	MoveL Offs(p0,26.0,100.0, 0), v10, z5, tool0;
	MoveL Offs(p0,27.0,102.0, 0), v10, z5, tool0;
	MoveL Offs(p0,27.0,104.0, 0), v10, z5, tool0;
	MoveL Offs(p0,27.0,107.0, 0), v10, z5, tool0;
	MoveL Offs(p0,27.0,109.0, 0), v10, z5, tool0;
	MoveL Offs(p0,27.0,110.0, 0), v10, z5, tool0;
	MoveL Offs(p0,26.0,112.0, 0), v10, z5, tool0;
	MoveL Offs(p0,26.0,113.0, 0), v10, z5, tool0;
	MoveL Offs(p0,29.0,114.0, 0), v10, z5, tool0;
	MoveJ Offs(p0,29.0,114.0, 20), v10, z1, tool0;
	MoveJ Offs(p0,123.0,112.0, 20), v10, z1, tool0;
	MoveJ Offs(p0,123.0,112.0, 0), v10, z1, tool0;
	MoveL Offs(p0,125.0,110.0, 0), v10, z5, tool0;
	MoveL Offs(p0,125.0,109.0, 0), v10, z5, tool0;
	MoveL Offs(p0,126.0,107.0, 0), v10, z5, tool0;
	MoveL Offs(p0,127.0,106.0, 0), v10, z5, tool0;
	MoveL Offs(p0,128.0,104.0, 0), v10, z5, tool0;
	MoveL Offs(p0,130.0,101.0, 0), v10, z5, tool0;
	MoveL Offs(p0,131.0,98.0, 0), v10, z5, tool0;
	MoveL Offs(p0,133.0,95.0, 0), v10, z5, tool0;
	MoveL Offs(p0,134.0,92.0, 0), v10, z5, tool0;
	MoveL Offs(p0,135.0,91.0, 0), v10, z5, tool0;
	MoveL Offs(p0,136.0,90.0, 0), v10, z5, tool0;
	MoveL Offs(p0,137.0,89.0, 0), v10, z5, tool0;
	MoveL Offs(p0,137.0,87.0, 0), v10, z5, tool0;
	MoveL Offs(p0,138.0,86.0, 0), v10, z5, tool0;
	MoveL Offs(p0,139.0,84.0, 0), v10, z5, tool0;
	MoveL Offs(p0,140.0,82.0, 0), v10, z5, tool0;
	MoveL Offs(p0,141.0,80.0, 0), v10, z5, tool0;
	MoveL Offs(p0,143.0,78.0, 0), v10, z5, tool0;
	MoveL Offs(p0,144.0,76.0, 0), v10, z5, tool0;
	MoveL Offs(p0,145.0,74.0, 0), v10, z5, tool0;
	MoveL Offs(p0,146.0,72.0, 0), v10, z5, tool0;
	MoveL Offs(p0,147.0,71.0, 0), v10, z5, tool0;
	MoveL Offs(p0,147.0,70.0, 0), v10, z5, tool0;
	MoveL Offs(p0,147.0,69.0, 0), v10, z5, tool0;
	MoveL Offs(p0,148.0,69.0, 0), v10, z5, tool0;
	MoveL Offs(p0,148.0,68.0, 0), v10, z5, tool0;
	MoveL Offs(p0,148.0,67.0, 0), v10, z5, tool0;
	MoveL Offs(p0,147.0,65.0, 0), v10, z5, tool0;
	MoveL Offs(p0,147.0,64.0, 0), v10, z5, tool0;
	MoveL Offs(p0,146.0,63.0, 0), v10, z5, tool0;
	MoveL Offs(p0,145.0,63.0, 0), v10, z5, tool0;
	MoveL Offs(p0,145.0,62.0, 0), v10, z5, tool0;
	MoveL Offs(p0,144.0,61.0, 0), v10, z5, tool0;
	MoveL Offs(p0,142.0,60.0, 0), v10, z5, tool0;
	MoveL Offs(p0,141.0,59.0, 0), v10, z5, tool0;
	MoveL Offs(p0,139.0,58.0, 0), v10, z5, tool0;
	MoveL Offs(p0,137.0,57.0, 0), v10, z5, tool0;
	MoveL Offs(p0,135.0,56.0, 0), v10, z5, tool0;
	MoveL Offs(p0,133.0,55.0, 0), v10, z5, tool0;
	MoveL Offs(p0,131.0,54.0, 0), v10, z5, tool0;
	MoveL Offs(p0,129.0,53.0, 0), v10, z5, tool0;
	MoveL Offs(p0,127.0,53.0, 0), v10, z5, tool0;
	MoveL Offs(p0,126.0,52.0, 0), v10, z5, tool0;
	MoveL Offs(p0,125.0,52.0, 0), v10, z5, tool0;
	MoveL Offs(p0,124.0,52.0, 0), v10, z5, tool0;
	MoveL Offs(p0,122.0,53.0, 0), v10, z5, tool0;
	MoveL Offs(p0,121.0,53.0, 0), v10, z5, tool0;
	MoveL Offs(p0,121.0,54.0, 0), v10, z5, tool0;
	MoveL Offs(p0,120.0,55.0, 0), v10, z5, tool0;
	MoveL Offs(p0,119.0,57.0, 0), v10, z5, tool0;
	MoveL Offs(p0,118.0,59.0, 0), v10, z5, tool0;
	MoveL Offs(p0,116.0,61.0, 0), v10, z5, tool0;
	MoveL Offs(p0,115.0,64.0, 0), v10, z5, tool0;
	MoveL Offs(p0,113.0,67.0, 0), v10, z5, tool0;
	MoveL Offs(p0,112.0,69.0, 0), v10, z5, tool0;
	MoveL Offs(p0,112.0,71.0, 0), v10, z5, tool0;
	MoveL Offs(p0,111.0,72.0, 0), v10, z5, tool0;
	MoveL Offs(p0,110.0,73.0, 0), v10, z5, tool0;
	MoveL Offs(p0,110.0,74.0, 0), v10, z5, tool0;
	MoveL Offs(p0,109.0,75.0, 0), v10, z5, tool0;
	MoveL Offs(p0,109.0,76.0, 0), v10, z5, tool0;
	MoveL Offs(p0,108.0,76.0, 0), v10, z5, tool0;
	MoveL Offs(p0,107.0,79.0, 0), v10, z5, tool0;
	MoveL Offs(p0,105.0,81.0, 0), v10, z5, tool0;
	MoveL Offs(p0,104.0,83.0, 0), v10, z5, tool0;
	MoveL Offs(p0,103.0,85.0, 0), v10, z5, tool0;
	MoveL Offs(p0,101.0,86.0, 0), v10, z5, tool0;
	MoveL Offs(p0,100.0,88.0, 0), v10, z5, tool0;
	MoveL Offs(p0,99.0,89.0, 0), v10, z5, tool0;
	MoveL Offs(p0,98.0,91.0, 0), v10, z5, tool0;
	MoveL Offs(p0,97.0,91.0, 0), v10, z5, tool0;
	MoveL Offs(p0,95.0,94.0, 0), v10, z5, tool0;
	MoveL Offs(p0,95.0,94.0, 0), v10, z5, tool0;
	MoveL Offs(p0,94.0,95.0, 0), v10, z5, tool0;
	MoveL Offs(p0,94.0,95.0, 0), v10, z5, tool0;
	MoveL Offs(p0,94.0,96.0, 0), v10, z5, tool0;
	MoveL Offs(p0,94.0,96.0, 0), v10, z5, tool0;
	MoveL Offs(p0,94.0,97.0, 0), v10, z5, tool0;
	MoveL Offs(p0,95.0,99.0, 0), v10, z5, tool0;
	MoveL Offs(p0,95.0,100.0, 0), v10, z5, tool0;
	MoveL Offs(p0,96.0,100.0, 0), v10, z5, tool0;
	MoveL Offs(p0,96.0,100.0, 0), v10, z5, tool0;
	MoveL Offs(p0,97.0,100.0, 0), v10, z5, tool0;
	MoveL Offs(p0,98.0,101.0, 0), v10, z5, tool0;
	MoveL Offs(p0,99.0,101.0, 0), v10, z5, tool0;
	MoveL Offs(p0,102.0,101.0, 0), v10, z5, tool0;
	MoveL Offs(p0,102.0,101.0, 0), v10, z5, tool0;
	MoveL Offs(p0,103.0,102.0, 0), v10, z5, tool0;
	MoveL Offs(p0,104.0,102.0, 0), v10, z5, tool0;
	MoveL Offs(p0,104.0,102.0, 0), v10, z5, tool0;
	MoveL Offs(p0,105.0,103.0, 0), v10, z5, tool0;
	MoveL Offs(p0,106.0,103.0, 0), v10, z5, tool0;
	MoveL Offs(p0,109.0,105.0, 0), v10, z5, tool0;
	MoveL Offs(p0,110.0,105.0, 0), v10, z5, tool0;
	MoveL Offs(p0,111.0,106.0, 0), v10, z5, tool0;
	MoveL Offs(p0,112.0,107.0, 0), v10, z5, tool0;
	MoveL Offs(p0,113.0,108.0, 0), v10, z5, tool0;
	MoveL Offs(p0,114.0,108.0, 0), v10, z5, tool0;
	MoveL Offs(p0,115.0,109.0, 0), v10, z5, tool0;
	MoveL Offs(p0,116.0,110.0, 0), v10, z5, tool0;
	MoveL Offs(p0,116.0,111.0, 0), v10, z5, tool0;
	MoveL Offs(p0,118.0,113.0, 0), v10, z5, tool0;
	MoveL Offs(p0,118.0,113.0, 0), v10, z5, tool0;
	MoveL Offs(p0,119.0,113.0, 0), v10, z5, tool0;
	MoveL Offs(p0,119.0,113.0, 0), v10, z5, tool0;
	MoveL Offs(p0,119.0,114.0, 0), v10, z5, tool0;
	MoveL Offs(p0,120.0,114.0, 0), v10, z5, tool0;
	MoveL Offs(p0,120.0,114.0, 0), v10, z5, tool0;
	MoveL Offs(p0,122.0,113.0, 0), v10, z5, tool0;
	MoveL Offs(p0,123.0,113.0, 0), v10, z5, tool0;
	MoveL Offs(p0,123.0,112.0, 0), v10, z5, tool0;
	MoveL Offs(p0,123.0,112.0, 0), v10, z5, tool0;
	MoveJ Offs(p0,123.0,112.0, 20), v10, z1, tool0;
	MoveJ Offs(p0,76.0,113.0, 20), v10, z1, tool0;
	MoveJ Offs(p0,76.0,113.0, 0), v10, z1, tool0;
	MoveL Offs(p0,75.0,109.0, 0), v10, z5, tool0;
	MoveL Offs(p0,74.0,109.0, 0), v10, z5, tool0;
	MoveL Offs(p0,74.0,108.0, 0), v10, z5, tool0;
	MoveL Offs(p0,73.0,107.0, 0), v10, z5, tool0;
	MoveL Offs(p0,72.0,107.0, 0), v10, z5, tool0;
	MoveL Offs(p0,71.0,106.0, 0), v10, z5, tool0;
	MoveL Offs(p0,69.0,104.0, 0), v10, z5, tool0;
	MoveL Offs(p0,69.0,104.0, 0), v10, z5, tool0;
	MoveL Offs(p0,68.0,104.0, 0), v10, z5, tool0;
	MoveL Offs(p0,68.0,104.0, 0), v10, z5, tool0;
	MoveL Offs(p0,67.0,104.0, 0), v10, z5, tool0;
	MoveL Offs(p0,67.0,104.0, 0), v10, z5, tool0;
	MoveL Offs(p0,67.0,105.0, 0), v10, z5, tool0;
	MoveL Offs(p0,66.0,105.0, 0), v10, z5, tool0;
	MoveL Offs(p0,65.0,106.0, 0), v10, z5, tool0;
	MoveL Offs(p0,69.0,109.0, 0), v10, z5, tool0;
	MoveL Offs(p0,71.0,111.0, 0), v10, z5, tool0;
	MoveL Offs(p0,72.0,112.0, 0), v10, z5, tool0;
	MoveL Offs(p0,72.0,112.0, 0), v10, z5, tool0;
	MoveL Offs(p0,72.0,112.0, 0), v10, z5, tool0;
	MoveL Offs(p0,73.0,113.0, 0), v10, z5, tool0;
	MoveL Offs(p0,73.0,113.0, 0), v10, z5, tool0;
	MoveL Offs(p0,73.0,113.0, 0), v10, z5, tool0;
	MoveL Offs(p0,76.0,113.0, 0), v10, z5, tool0;
	MoveJ Offs(p0,76.0,113.0, 20), v10, z1, tool0;
	MoveJ Offs(p0,116.0,113.0, 20), v10, z1, tool0;
	MoveJ Offs(p0,116.0,113.0, 0), v10, z1, tool0;
	MoveL Offs(p0,115.0,111.0, 0), v10, z5, tool0;
	MoveL Offs(p0,114.0,110.0, 0), v10, z5, tool0;
	MoveL Offs(p0,114.0,109.0, 0), v10, z5, tool0;
	MoveL Offs(p0,113.0,109.0, 0), v10, z5, tool0;
	MoveL Offs(p0,113.0,108.0, 0), v10, z5, tool0;
	MoveL Offs(p0,112.0,108.0, 0), v10, z5, tool0;
	MoveL Offs(p0,110.0,106.0, 0), v10, z5, tool0;
	MoveL Offs(p0,109.0,106.0, 0), v10, z5, tool0;
	MoveL Offs(p0,109.0,106.0, 0), v10, z5, tool0;
	MoveL Offs(p0,108.0,105.0, 0), v10, z5, tool0;
	MoveL Offs(p0,107.0,105.0, 0), v10, z5, tool0;
	MoveL Offs(p0,107.0,105.0, 0), v10, z5, tool0;
	MoveL Offs(p0,104.0,103.0, 0), v10, z5, tool0;
	MoveL Offs(p0,104.0,103.0, 0), v10, z5, tool0;
	MoveL Offs(p0,103.0,103.0, 0), v10, z5, tool0;
	MoveL Offs(p0,102.0,103.0, 0), v10, z5, tool0;
	MoveL Offs(p0,102.0,102.0, 0), v10, z5, tool0;
	MoveL Offs(p0,101.0,102.0, 0), v10, z5, tool0;
	MoveL Offs(p0,101.0,102.0, 0), v10, z5, tool0;
	MoveL Offs(p0,100.0,102.0, 0), v10, z5, tool0;
	MoveL Offs(p0,98.0,102.0, 0), v10, z5, tool0;
	MoveL Offs(p0,98.0,102.0, 0), v10, z5, tool0;
	MoveL Offs(p0,97.0,102.0, 0), v10, z5, tool0;
	MoveL Offs(p0,97.0,102.0, 0), v10, z5, tool0;
	MoveL Offs(p0,97.0,102.0, 0), v10, z5, tool0;
	MoveL Offs(p0,97.0,102.0, 0), v10, z5, tool0;
	MoveL Offs(p0,96.0,101.0, 0), v10, z5, tool0;
	MoveL Offs(p0,96.0,103.0, 0), v10, z5, tool0;
	MoveL Offs(p0,97.0,105.0, 0), v10, z5, tool0;
	MoveL Offs(p0,97.0,106.0, 0), v10, z5, tool0;
	MoveL Offs(p0,97.0,106.0, 0), v10, z5, tool0;
	MoveL Offs(p0,97.0,106.0, 0), v10, z5, tool0;
	MoveL Offs(p0,97.0,106.0, 0), v10, z5, tool0;
	MoveL Offs(p0,98.0,107.0, 0), v10, z5, tool0;
	MoveL Offs(p0,100.0,107.0, 0), v10, z5, tool0;
	MoveL Offs(p0,100.0,107.0, 0), v10, z5, tool0;
	MoveL Offs(p0,101.0,107.0, 0), v10, z5, tool0;
	MoveL Offs(p0,101.0,107.0, 0), v10, z5, tool0;
	MoveL Offs(p0,103.0,107.0, 0), v10, z5, tool0;
	MoveL Offs(p0,104.0,107.0, 0), v10, z5, tool0;
	MoveL Offs(p0,105.0,107.0, 0), v10, z5, tool0;
	MoveL Offs(p0,105.0,107.0, 0), v10, z5, tool0;
	MoveL Offs(p0,106.0,108.0, 0), v10, z5, tool0;
	MoveL Offs(p0,106.0,108.0, 0), v10, z5, tool0;
	MoveL Offs(p0,107.0,109.0, 0), v10, z5, tool0;
	MoveL Offs(p0,107.0,110.0, 0), v10, z5, tool0;
	MoveL Offs(p0,108.0,111.0, 0), v10, z5, tool0;
	MoveL Offs(p0,109.0,113.0, 0), v10, z5, tool0;
	MoveL Offs(p0,112.0,113.0, 0), v10, z5, tool0;
	MoveL Offs(p0,114.0,113.0, 0), v10, z5, tool0;
	MoveL Offs(p0,115.0,113.0, 0), v10, z5, tool0;
	MoveL Offs(p0,115.0,113.0, 0), v10, z5, tool0;
	MoveL Offs(p0,115.0,113.0, 0), v10, z5, tool0;
	MoveL Offs(p0,116.0,113.0, 0), v10, z5, tool0;
	MoveL Offs(p0,116.0,113.0, 0), v10, z5, tool0;
	MoveL Offs(p0,116.0,113.0, 0), v10, z5, tool0;
	MoveL Offs(p0,116.0,113.0, 0), v10, z5, tool0;
	MoveJ Offs(p0,116.0,113.0, 20), v10, z1, tool0;
	MoveJ Offs(p0,82.0,111.0, 20), v10, z1, tool0;
	MoveJ Offs(p0,82.0,111.0, 0), v10, z1, tool0;
	MoveL Offs(p0,84.0,110.0, 0), v10, z5, tool0;
	MoveL Offs(p0,84.0,109.0, 0), v10, z5, tool0;
	MoveL Offs(p0,85.0,109.0, 0), v10, z5, tool0;
	MoveL Offs(p0,86.0,106.0, 0), v10, z5, tool0;
	MoveL Offs(p0,87.0,105.0, 0), v10, z5, tool0;
	MoveL Offs(p0,88.0,104.0, 0), v10, z5, tool0;
	MoveL Offs(p0,89.0,103.0, 0), v10, z5, tool0;
	MoveL Offs(p0,90.0,103.0, 0), v10, z5, tool0;
	MoveL Offs(p0,91.0,102.0, 0), v10, z5, tool0;
	MoveL Offs(p0,92.0,102.0, 0), v10, z5, tool0;
	MoveL Offs(p0,93.0,102.0, 0), v10, z5, tool0;
	MoveL Offs(p0,94.0,102.0, 0), v10, z5, tool0;
	MoveL Offs(p0,94.0,100.0, 0), v10, z5, tool0;
	MoveL Offs(p0,94.0,100.0, 0), v10, z5, tool0;
	MoveL Offs(p0,93.0,98.0, 0), v10, z5, tool0;
	MoveL Offs(p0,93.0,97.0, 0), v10, z5, tool0;
	MoveL Offs(p0,93.0,96.0, 0), v10, z5, tool0;
	MoveL Offs(p0,93.0,96.0, 0), v10, z5, tool0;
	MoveL Offs(p0,93.0,95.0, 0), v10, z5, tool0;
	MoveL Offs(p0,93.0,95.0, 0), v10, z5, tool0;
	MoveL Offs(p0,93.0,94.0, 0), v10, z5, tool0;
	MoveL Offs(p0,95.0,92.0, 0), v10, z5, tool0;
	MoveL Offs(p0,95.0,91.0, 0), v10, z5, tool0;
	MoveL Offs(p0,96.0,91.0, 0), v10, z5, tool0;
	MoveL Offs(p0,96.0,90.0, 0), v10, z5, tool0;
	MoveL Offs(p0,97.0,90.0, 0), v10, z5, tool0;
	MoveL Offs(p0,99.0,88.0, 0), v10, z5, tool0;
	MoveL Offs(p0,99.0,87.0, 0), v10, z5, tool0;
	MoveL Offs(p0,100.0,86.0, 0), v10, z5, tool0;
	MoveL Offs(p0,101.0,86.0, 0), v10, z5, tool0;
	MoveL Offs(p0,101.0,85.0, 0), v10, z5, tool0;
	MoveL Offs(p0,102.0,84.0, 0), v10, z5, tool0;
	MoveL Offs(p0,102.0,84.0, 0), v10, z5, tool0;
	MoveL Offs(p0,102.0,83.0, 0), v10, z5, tool0;
	MoveL Offs(p0,95.0,86.0, 0), v10, z5, tool0;
	MoveL Offs(p0,95.0,86.0, 0), v10, z5, tool0;
	MoveL Offs(p0,94.0,86.0, 0), v10, z5, tool0;
	MoveL Offs(p0,93.0,86.0, 0), v10, z5, tool0;
	MoveL Offs(p0,93.0,86.0, 0), v10, z5, tool0;
	MoveL Offs(p0,92.0,86.0, 0), v10, z5, tool0;
	MoveL Offs(p0,92.0,85.0, 0), v10, z5, tool0;
	MoveL Offs(p0,89.0,85.0, 0), v10, z5, tool0;
	MoveL Offs(p0,88.0,84.0, 0), v10, z5, tool0;
	MoveL Offs(p0,87.0,84.0, 0), v10, z5, tool0;
	MoveL Offs(p0,87.0,84.0, 0), v10, z5, tool0;
	MoveL Offs(p0,86.0,84.0, 0), v10, z5, tool0;
	MoveL Offs(p0,86.0,84.0, 0), v10, z5, tool0;
	MoveL Offs(p0,85.0,85.0, 0), v10, z5, tool0;
	MoveL Offs(p0,85.0,85.0, 0), v10, z5, tool0;
	MoveL Offs(p0,84.0,86.0, 0), v10, z5, tool0;
	MoveL Offs(p0,84.0,87.0, 0), v10, z5, tool0;
	MoveL Offs(p0,85.0,88.0, 0), v10, z5, tool0;
	MoveL Offs(p0,86.0,90.0, 0), v10, z5, tool0;
	MoveL Offs(p0,86.0,91.0, 0), v10, z5, tool0;
	MoveL Offs(p0,86.0,91.0, 0), v10, z5, tool0;
	MoveL Offs(p0,86.0,92.0, 0), v10, z5, tool0;
	MoveL Offs(p0,86.0,92.0, 0), v10, z5, tool0;
	MoveL Offs(p0,85.0,93.0, 0), v10, z5, tool0;
	MoveL Offs(p0,84.0,95.0, 0), v10, z5, tool0;
	MoveL Offs(p0,83.0,96.0, 0), v10, z5, tool0;
	MoveL Offs(p0,82.0,96.0, 0), v10, z5, tool0;
	MoveL Offs(p0,81.0,97.0, 0), v10, z5, tool0;
	MoveL Offs(p0,79.0,97.0, 0), v10, z5, tool0;
	MoveL Offs(p0,78.0,97.0, 0), v10, z5, tool0;
	MoveL Offs(p0,76.0,97.0, 0), v10, z5, tool0;
	MoveL Offs(p0,74.0,97.0, 0), v10, z5, tool0;
	MoveL Offs(p0,72.0,97.0, 0), v10, z5, tool0;
	MoveL Offs(p0,68.0,96.0, 0), v10, z5, tool0;
	MoveL Offs(p0,67.0,97.0, 0), v10, z5, tool0;
	MoveL Offs(p0,66.0,99.0, 0), v10, z5, tool0;
	MoveL Offs(p0,66.0,100.0, 0), v10, z5, tool0;
	MoveL Offs(p0,66.0,100.0, 0), v10, z5, tool0;
	MoveL Offs(p0,67.0,101.0, 0), v10, z5, tool0;
	MoveL Offs(p0,67.0,101.0, 0), v10, z5, tool0;
	MoveL Offs(p0,68.0,102.0, 0), v10, z5, tool0;
	MoveL Offs(p0,70.0,103.0, 0), v10, z5, tool0;
	MoveL Offs(p0,71.0,104.0, 0), v10, z5, tool0;
	MoveL Offs(p0,73.0,105.0, 0), v10, z5, tool0;
	MoveL Offs(p0,74.0,106.0, 0), v10, z5, tool0;
	MoveL Offs(p0,75.0,108.0, 0), v10, z5, tool0;
	MoveL Offs(p0,76.0,109.0, 0), v10, z5, tool0;
	MoveL Offs(p0,77.0,110.0, 0), v10, z5, tool0;
	MoveL Offs(p0,77.0,110.0, 0), v10, z5, tool0;
	MoveL Offs(p0,78.0,111.0, 0), v10, z5, tool0;
	MoveL Offs(p0,82.0,111.0, 0), v10, z5, tool0;
	MoveL Offs(p0,82.0,111.0, 0), v10, z5, tool0;
	MoveL Offs(p0,82.0,111.0, 0), v10, z5, tool0;
	MoveJ Offs(p0,82.0,111.0, 20), v10, z1, tool0;
	MoveJ Offs(p0,62.0,110.0, 20), v10, z1, tool0;
	MoveJ Offs(p0,62.0,110.0, 0), v10, z1, tool0;
	MoveL Offs(p0,63.0,108.0, 0), v10, z5, tool0;
	MoveL Offs(p0,64.0,107.0, 0), v10, z5, tool0;
	MoveL Offs(p0,64.0,107.0, 0), v10, z5, tool0;
	MoveL Offs(p0,64.0,107.0, 0), v10, z5, tool0;
	MoveL Offs(p0,64.0,106.0, 0), v10, z5, tool0;
	MoveL Offs(p0,66.0,104.0, 0), v10, z5, tool0;
	MoveL Offs(p0,66.0,104.0, 0), v10, z5, tool0;
	MoveL Offs(p0,66.0,103.0, 0), v10, z5, tool0;
	MoveL Offs(p0,66.0,103.0, 0), v10, z5, tool0;
	MoveL Offs(p0,66.0,103.0, 0), v10, z5, tool0;
	MoveL Offs(p0,66.0,103.0, 0), v10, z5, tool0;
	MoveL Offs(p0,64.0,99.0, 0), v10, z5, tool0;
	MoveL Offs(p0,65.0,99.0, 0), v10, z5, tool0;
	MoveL Offs(p0,65.0,98.0, 0), v10, z5, tool0;
	MoveL Offs(p0,65.0,98.0, 0), v10, z5, tool0;
	MoveL Offs(p0,65.0,97.0, 0), v10, z5, tool0;
	MoveL Offs(p0,66.0,95.0, 0), v10, z5, tool0;
	MoveL Offs(p0,66.0,95.0, 0), v10, z5, tool0;
	MoveL Offs(p0,65.0,94.0, 0), v10, z5, tool0;
	MoveL Offs(p0,65.0,94.0, 0), v10, z5, tool0;
	MoveL Offs(p0,65.0,94.0, 0), v10, z5, tool0;
	MoveL Offs(p0,64.0,94.0, 0), v10, z5, tool0;
	MoveL Offs(p0,62.0,94.0, 0), v10, z5, tool0;
	MoveL Offs(p0,62.0,94.0, 0), v10, z5, tool0;
	MoveL Offs(p0,62.0,94.0, 0), v10, z5, tool0;
	MoveL Offs(p0,60.0,97.0, 0), v10, z5, tool0;
	MoveL Offs(p0,60.0,98.0, 0), v10, z5, tool0;
	MoveL Offs(p0,60.0,99.0, 0), v10, z5, tool0;
	MoveL Offs(p0,60.0,100.0, 0), v10, z5, tool0;
	MoveL Offs(p0,60.0,101.0, 0), v10, z5, tool0;
	MoveL Offs(p0,60.0,102.0, 0), v10, z5, tool0;
	MoveL Offs(p0,60.0,103.0, 0), v10, z5, tool0;
	MoveL Offs(p0,60.0,105.0, 0), v10, z5, tool0;
	MoveL Offs(p0,60.0,106.0, 0), v10, z5, tool0;
	MoveL Offs(p0,60.0,108.0, 0), v10, z5, tool0;
	MoveL Offs(p0,60.0,109.0, 0), v10, z5, tool0;
	MoveL Offs(p0,60.0,109.0, 0), v10, z5, tool0;
	MoveL Offs(p0,61.0,110.0, 0), v10, z5, tool0;
	MoveL Offs(p0,61.0,111.0, 0), v10, z5, tool0;
	MoveL Offs(p0,61.0,111.0, 0), v10, z5, tool0;
	MoveL Offs(p0,61.0,111.0, 0), v10, z5, tool0;
	MoveL Offs(p0,62.0,110.0, 0), v10, z5, tool0;
	MoveJ Offs(p0,62.0,110.0, 20), v10, z1, tool0;
	MoveJ Offs(p0,92.0,108.0, 20), v10, z1, tool0;
	MoveJ Offs(p0,92.0,108.0, 0), v10, z1, tool0;
	MoveL Offs(p0,93.0,106.0, 0), v10, z5, tool0;
	MoveL Offs(p0,93.0,106.0, 0), v10, z5, tool0;
	MoveL Offs(p0,93.0,106.0, 0), v10, z5, tool0;
	MoveL Offs(p0,91.0,103.0, 0), v10, z5, tool0;
	MoveL Offs(p0,89.0,105.0, 0), v10, z5, tool0;
	MoveL Offs(p0,88.0,106.0, 0), v10, z5, tool0;
	MoveL Offs(p0,88.0,106.0, 0), v10, z5, tool0;
	MoveL Offs(p0,87.0,107.0, 0), v10, z5, tool0;
	MoveL Offs(p0,87.0,107.0, 0), v10, z5, tool0;
	MoveL Offs(p0,86.0,108.0, 0), v10, z5, tool0;
	MoveL Offs(p0,85.0,110.0, 0), v10, z5, tool0;
	MoveL Offs(p0,86.0,110.0, 0), v10, z5, tool0;
	MoveL Offs(p0,86.0,110.0, 0), v10, z5, tool0;
	MoveL Offs(p0,87.0,110.0, 0), v10, z5, tool0;
	MoveL Offs(p0,87.0,110.0, 0), v10, z5, tool0;
	MoveL Offs(p0,91.0,110.0, 0), v10, z5, tool0;
	MoveL Offs(p0,91.0,109.0, 0), v10, z5, tool0;
	MoveL Offs(p0,91.0,109.0, 0), v10, z5, tool0;
	MoveL Offs(p0,91.0,109.0, 0), v10, z5, tool0;
	MoveL Offs(p0,91.0,109.0, 0), v10, z5, tool0;
	MoveL Offs(p0,91.0,109.0, 0), v10, z5, tool0;
	MoveL Offs(p0,92.0,108.0, 0), v10, z5, tool0;
	MoveL Offs(p0,92.0,108.0, 0), v10, z5, tool0;
	MoveJ Offs(p0,92.0,108.0, 20), v10, z1, tool0;
	MoveJ Offs(p0,146.0,98.0, 20), v10, z1, tool0;
	MoveJ Offs(p0,146.0,98.0, 0), v10, z1, tool0;
	MoveL Offs(p0,148.0,96.0, 0), v10, z5, tool0;
	MoveL Offs(p0,149.0,95.0, 0), v10, z5, tool0;
	MoveL Offs(p0,150.0,94.0, 0), v10, z5, tool0;
	MoveL Offs(p0,150.0,94.0, 0), v10, z5, tool0;
	MoveL Offs(p0,151.0,93.0, 0), v10, z5, tool0;
	MoveL Offs(p0,151.0,92.0, 0), v10, z5, tool0;
	MoveL Offs(p0,152.0,90.0, 0), v10, z5, tool0;
	MoveL Offs(p0,152.0,89.0, 0), v10, z5, tool0;
	MoveL Offs(p0,153.0,86.0, 0), v10, z5, tool0;
	MoveL Offs(p0,154.0,83.0, 0), v10, z5, tool0;
	MoveL Offs(p0,155.0,81.0, 0), v10, z5, tool0;
	MoveL Offs(p0,156.0,79.0, 0), v10, z5, tool0;
	MoveL Offs(p0,157.0,77.0, 0), v10, z5, tool0;
	MoveL Offs(p0,158.0,75.0, 0), v10, z5, tool0;
	MoveL Offs(p0,159.0,74.0, 0), v10, z5, tool0;
	MoveL Offs(p0,161.0,73.0, 0), v10, z5, tool0;
	MoveL Offs(p0,162.0,71.0, 0), v10, z5, tool0;
	MoveL Offs(p0,163.0,70.0, 0), v10, z5, tool0;
	MoveL Offs(p0,166.0,69.0, 0), v10, z5, tool0;
	MoveL Offs(p0,167.0,69.0, 0), v10, z5, tool0;
	MoveL Offs(p0,168.0,68.0, 0), v10, z5, tool0;
	MoveL Offs(p0,170.0,68.0, 0), v10, z5, tool0;
	MoveL Offs(p0,171.0,68.0, 0), v10, z5, tool0;
	MoveL Offs(p0,173.0,68.0, 0), v10, z5, tool0;
	MoveL Offs(p0,174.0,68.0, 0), v10, z5, tool0;
	MoveL Offs(p0,176.0,68.0, 0), v10, z5, tool0;
	MoveL Offs(p0,177.0,68.0, 0), v10, z5, tool0;
	MoveL Offs(p0,180.0,69.0, 0), v10, z5, tool0;
	MoveL Offs(p0,182.0,70.0, 0), v10, z5, tool0;
	MoveL Offs(p0,183.0,71.0, 0), v10, z5, tool0;
	MoveL Offs(p0,184.0,73.0, 0), v10, z5, tool0;
	MoveL Offs(p0,184.0,74.0, 0), v10, z5, tool0;
	MoveL Offs(p0,185.0,75.0, 0), v10, z5, tool0;
	MoveL Offs(p0,185.0,77.0, 0), v10, z5, tool0;
	MoveL Offs(p0,185.0,79.0, 0), v10, z5, tool0;
	MoveL Offs(p0,184.0,80.0, 0), v10, z5, tool0;
	MoveL Offs(p0,182.0,84.0, 0), v10, z5, tool0;
	MoveL Offs(p0,181.0,86.0, 0), v10, z5, tool0;
	MoveL Offs(p0,180.0,87.0, 0), v10, z5, tool0;
	MoveL Offs(p0,178.0,88.0, 0), v10, z5, tool0;
	MoveL Offs(p0,176.0,89.0, 0), v10, z5, tool0;
	MoveL Offs(p0,174.0,90.0, 0), v10, z5, tool0;
	MoveL Offs(p0,172.0,91.0, 0), v10, z5, tool0;
	MoveL Offs(p0,170.0,91.0, 0), v10, z5, tool0;
	MoveL Offs(p0,167.0,91.0, 0), v10, z5, tool0;
	MoveL Offs(p0,165.0,91.0, 0), v10, z5, tool0;
	MoveL Offs(p0,165.0,91.0, 0), v10, z5, tool0;
	MoveL Offs(p0,165.0,91.0, 0), v10, z5, tool0;
	MoveL Offs(p0,164.0,91.0, 0), v10, z5, tool0;
	MoveL Offs(p0,164.0,91.0, 0), v10, z5, tool0;
	MoveL Offs(p0,164.0,91.0, 0), v10, z5, tool0;
	MoveL Offs(p0,167.0,92.0, 0), v10, z5, tool0;
	MoveL Offs(p0,167.0,92.0, 0), v10, z5, tool0;
	MoveL Offs(p0,168.0,92.0, 0), v10, z5, tool0;
	MoveL Offs(p0,168.0,92.0, 0), v10, z5, tool0;
	MoveL Offs(p0,169.0,92.0, 0), v10, z5, tool0;
	MoveL Offs(p0,171.0,92.0, 0), v10, z5, tool0;
	MoveL Offs(p0,172.0,92.0, 0), v10, z5, tool0;
	MoveL Offs(p0,173.0,92.0, 0), v10, z5, tool0;
	MoveL Offs(p0,173.0,92.0, 0), v10, z5, tool0;
	MoveL Offs(p0,174.0,91.0, 0), v10, z5, tool0;
	MoveL Offs(p0,174.0,91.0, 0), v10, z5, tool0;
	MoveL Offs(p0,175.0,91.0, 0), v10, z5, tool0;
	MoveL Offs(p0,176.0,91.0, 0), v10, z5, tool0;
	MoveL Offs(p0,177.0,90.0, 0), v10, z5, tool0;
	MoveL Offs(p0,179.0,89.0, 0), v10, z5, tool0;
	MoveL Offs(p0,180.0,88.0, 0), v10, z5, tool0;
	MoveL Offs(p0,181.0,87.0, 0), v10, z5, tool0;
	MoveL Offs(p0,182.0,87.0, 0), v10, z5, tool0;
	MoveL Offs(p0,183.0,86.0, 0), v10, z5, tool0;
	MoveL Offs(p0,184.0,85.0, 0), v10, z5, tool0;
	MoveL Offs(p0,184.0,84.0, 0), v10, z5, tool0;
	MoveL Offs(p0,185.0,83.0, 0), v10, z5, tool0;
	MoveL Offs(p0,186.0,82.0, 0), v10, z5, tool0;
	MoveL Offs(p0,187.0,79.0, 0), v10, z5, tool0;
	MoveL Offs(p0,187.0,79.0, 0), v10, z5, tool0;
	MoveL Offs(p0,187.0,78.0, 0), v10, z5, tool0;
	MoveL Offs(p0,187.0,77.0, 0), v10, z5, tool0;
	MoveL Offs(p0,187.0,76.0, 0), v10, z5, tool0;
	MoveL Offs(p0,187.0,75.0, 0), v10, z5, tool0;
	MoveL Offs(p0,187.0,74.0, 0), v10, z5, tool0;
	MoveL Offs(p0,187.0,74.0, 0), v10, z5, tool0;
	MoveL Offs(p0,186.0,71.0, 0), v10, z5, tool0;
	MoveL Offs(p0,185.0,70.0, 0), v10, z5, tool0;
	MoveL Offs(p0,184.0,70.0, 0), v10, z5, tool0;
	MoveL Offs(p0,184.0,69.0, 0), v10, z5, tool0;
	MoveL Offs(p0,183.0,68.0, 0), v10, z5, tool0;
	MoveL Offs(p0,182.0,68.0, 0), v10, z5, tool0;
	MoveL Offs(p0,181.0,67.0, 0), v10, z5, tool0;
	MoveL Offs(p0,181.0,67.0, 0), v10, z5, tool0;
	MoveL Offs(p0,178.0,66.0, 0), v10, z5, tool0;
	MoveL Offs(p0,178.0,66.0, 0), v10, z5, tool0;
	MoveL Offs(p0,177.0,65.0, 0), v10, z5, tool0;
	MoveL Offs(p0,177.0,65.0, 0), v10, z5, tool0;
	MoveL Offs(p0,176.0,65.0, 0), v10, z5, tool0;
	MoveL Offs(p0,175.0,65.0, 0), v10, z5, tool0;
	MoveL Offs(p0,174.0,65.0, 0), v10, z5, tool0;
	MoveL Offs(p0,172.0,65.0, 0), v10, z5, tool0;
	MoveL Offs(p0,171.0,65.0, 0), v10, z5, tool0;
	MoveL Offs(p0,171.0,65.0, 0), v10, z5, tool0;
	MoveL Offs(p0,170.0,65.0, 0), v10, z5, tool0;
	MoveL Offs(p0,170.0,65.0, 0), v10, z5, tool0;
	MoveL Offs(p0,169.0,66.0, 0), v10, z5, tool0;
	MoveL Offs(p0,168.0,66.0, 0), v10, z5, tool0;
	MoveL Offs(p0,168.0,66.0, 0), v10, z5, tool0;
	MoveL Offs(p0,165.0,67.0, 0), v10, z5, tool0;
	MoveL Offs(p0,163.0,68.0, 0), v10, z5, tool0;
	MoveL Offs(p0,161.0,69.0, 0), v10, z5, tool0;
	MoveL Offs(p0,159.0,71.0, 0), v10, z5, tool0;
	MoveL Offs(p0,158.0,73.0, 0), v10, z5, tool0;
	MoveL Offs(p0,156.0,75.0, 0), v10, z5, tool0;
	MoveL Offs(p0,154.0,77.0, 0), v10, z5, tool0;
	MoveL Offs(p0,153.0,80.0, 0), v10, z5, tool0;
	MoveL Offs(p0,152.0,83.0, 0), v10, z5, tool0;
	MoveL Offs(p0,151.0,86.0, 0), v10, z5, tool0;
	MoveL Offs(p0,150.0,88.0, 0), v10, z5, tool0;
	MoveL Offs(p0,150.0,89.0, 0), v10, z5, tool0;
	MoveL Offs(p0,149.0,90.0, 0), v10, z5, tool0;
	MoveL Offs(p0,149.0,90.0, 0), v10, z5, tool0;
	MoveL Offs(p0,149.0,91.0, 0), v10, z5, tool0;
	MoveL Offs(p0,149.0,91.0, 0), v10, z5, tool0;
	MoveL Offs(p0,149.0,92.0, 0), v10, z5, tool0;
	MoveL Offs(p0,148.0,92.0, 0), v10, z5, tool0;
	MoveL Offs(p0,147.0,94.0, 0), v10, z5, tool0;
	MoveL Offs(p0,146.0,95.0, 0), v10, z5, tool0;
	MoveL Offs(p0,145.0,96.0, 0), v10, z5, tool0;
	MoveL Offs(p0,143.0,96.0, 0), v10, z5, tool0;
	MoveL Offs(p0,142.0,97.0, 0), v10, z5, tool0;
	MoveL Offs(p0,141.0,97.0, 0), v10, z5, tool0;
	MoveL Offs(p0,140.0,97.0, 0), v10, z5, tool0;
	MoveL Offs(p0,138.0,97.0, 0), v10, z5, tool0;
	MoveL Offs(p0,137.0,97.0, 0), v10, z5, tool0;
	MoveL Offs(p0,135.0,96.0, 0), v10, z5, tool0;
	MoveL Offs(p0,135.0,97.0, 0), v10, z5, tool0;
	MoveL Offs(p0,139.0,99.0, 0), v10, z5, tool0;
	MoveL Offs(p0,140.0,99.0, 0), v10, z5, tool0;
	MoveL Offs(p0,141.0,99.0, 0), v10, z5, tool0;
	MoveL Offs(p0,142.0,99.0, 0), v10, z5, tool0;
	MoveL Offs(p0,143.0,99.0, 0), v10, z5, tool0;
	MoveL Offs(p0,144.0,99.0, 0), v10, z5, tool0;
	MoveL Offs(p0,145.0,98.0, 0), v10, z5, tool0;
	MoveL Offs(p0,146.0,98.0, 0), v10, z5, tool0;
	MoveL Offs(p0,146.0,98.0, 0), v10, z5, tool0;
	MoveJ Offs(p0,146.0,98.0, 20), v10, z1, tool0;
	MoveJ Offs(p0,81.0,96.0, 20), v10, z1, tool0;
	MoveJ Offs(p0,81.0,96.0, 0), v10, z1, tool0;
	MoveL Offs(p0,83.0,94.0, 0), v10, z5, tool0;
	MoveL Offs(p0,83.0,93.0, 0), v10, z5, tool0;
	MoveL Offs(p0,84.0,93.0, 0), v10, z5, tool0;
	MoveL Offs(p0,84.0,93.0, 0), v10, z5, tool0;
	MoveL Offs(p0,84.0,92.0, 0), v10, z5, tool0;
	MoveL Offs(p0,82.0,92.0, 0), v10, z5, tool0;
	MoveL Offs(p0,81.0,92.0, 0), v10, z5, tool0;
	MoveL Offs(p0,78.0,92.0, 0), v10, z5, tool0;
	MoveL Offs(p0,76.0,92.0, 0), v10, z5, tool0;
	MoveL Offs(p0,74.0,91.0, 0), v10, z5, tool0;
	MoveL Offs(p0,72.0,91.0, 0), v10, z5, tool0;
	MoveL Offs(p0,70.0,91.0, 0), v10, z5, tool0;
	MoveL Offs(p0,67.0,90.0, 0), v10, z5, tool0;
	MoveL Offs(p0,65.0,89.0, 0), v10, z5, tool0;
	MoveL Offs(p0,62.0,89.0, 0), v10, z5, tool0;
	MoveL Offs(p0,59.0,88.0, 0), v10, z5, tool0;
	MoveL Offs(p0,57.0,87.0, 0), v10, z5, tool0;
	MoveL Offs(p0,54.0,86.0, 0), v10, z5, tool0;
	MoveL Offs(p0,51.0,85.0, 0), v10, z5, tool0;
	MoveL Offs(p0,48.0,84.0, 0), v10, z5, tool0;
	MoveL Offs(p0,46.0,83.0, 0), v10, z5, tool0;
	MoveL Offs(p0,44.0,82.0, 0), v10, z5, tool0;
	MoveL Offs(p0,41.0,81.0, 0), v10, z5, tool0;
	MoveL Offs(p0,40.0,80.0, 0), v10, z5, tool0;
	MoveL Offs(p0,38.0,79.0, 0), v10, z5, tool0;
	MoveL Offs(p0,37.0,78.0, 0), v10, z5, tool0;
	MoveL Offs(p0,35.0,77.0, 0), v10, z5, tool0;
	MoveL Offs(p0,35.0,77.0, 0), v10, z5, tool0;
	MoveL Offs(p0,35.0,78.0, 0), v10, z5, tool0;
	MoveL Offs(p0,37.0,82.0, 0), v10, z5, tool0;
	MoveL Offs(p0,39.0,83.0, 0), v10, z5, tool0;
	MoveL Offs(p0,42.0,84.0, 0), v10, z5, tool0;
	MoveL Offs(p0,46.0,86.0, 0), v10, z5, tool0;
	MoveL Offs(p0,50.0,88.0, 0), v10, z5, tool0;
	MoveL Offs(p0,55.0,89.0, 0), v10, z5, tool0;
	MoveL Offs(p0,59.0,91.0, 0), v10, z5, tool0;
	MoveL Offs(p0,63.0,92.0, 0), v10, z5, tool0;
	MoveL Offs(p0,67.0,94.0, 0), v10, z5, tool0;
	MoveL Offs(p0,70.0,94.0, 0), v10, z5, tool0;
	MoveL Offs(p0,72.0,95.0, 0), v10, z5, tool0;
	MoveL Offs(p0,73.0,95.0, 0), v10, z5, tool0;
	MoveL Offs(p0,75.0,96.0, 0), v10, z5, tool0;
	MoveL Offs(p0,76.0,96.0, 0), v10, z5, tool0;
	MoveL Offs(p0,77.0,96.0, 0), v10, z5, tool0;
	MoveL Offs(p0,78.0,96.0, 0), v10, z5, tool0;
	MoveL Offs(p0,79.0,96.0, 0), v10, z5, tool0;
	MoveL Offs(p0,80.0,96.0, 0), v10, z5, tool0;
	MoveL Offs(p0,81.0,96.0, 0), v10, z5, tool0;
	MoveL Offs(p0,81.0,96.0, 0), v10, z5, tool0;
	MoveJ Offs(p0,81.0,96.0, 20), v10, z1, tool0;
	MoveJ Offs(p0,67.0,95.0, 20), v10, z1, tool0;
	MoveJ Offs(p0,67.0,95.0, 0), v10, z1, tool0;
	MoveL Offs(p0,67.0,95.0, 0), v10, z5, tool0;
	MoveJ Offs(p0,67.0,95.0, 20), v10, z1, tool0;
	MoveJ Offs(p0,21.0,90.0, 20), v10, z1, tool0;
	MoveJ Offs(p0,21.0,90.0, 0), v10, z1, tool0;
	MoveL Offs(p0,23.0,88.0, 0), v10, z5, tool0;
	MoveL Offs(p0,23.0,88.0, 0), v10, z5, tool0;
	MoveL Offs(p0,24.0,85.0, 0), v10, z5, tool0;
	MoveL Offs(p0,24.0,84.0, 0), v10, z5, tool0;
	MoveL Offs(p0,24.0,82.0, 0), v10, z5, tool0;
	MoveL Offs(p0,23.0,81.0, 0), v10, z5, tool0;
	MoveL Offs(p0,23.0,80.0, 0), v10, z5, tool0;
	MoveL Offs(p0,22.0,78.0, 0), v10, z5, tool0;
	MoveL Offs(p0,22.0,77.0, 0), v10, z5, tool0;
	MoveL Offs(p0,21.0,76.0, 0), v10, z5, tool0;
	MoveL Offs(p0,18.0,78.0, 0), v10, z5, tool0;
	MoveL Offs(p0,16.0,80.0, 0), v10, z5, tool0;
	MoveL Offs(p0,15.0,80.0, 0), v10, z5, tool0;
	MoveL Offs(p0,14.0,81.0, 0), v10, z5, tool0;
	MoveL Offs(p0,14.0,81.0, 0), v10, z5, tool0;
	MoveL Offs(p0,13.0,81.0, 0), v10, z5, tool0;
	MoveL Offs(p0,12.0,81.0, 0), v10, z5, tool0;
	MoveL Offs(p0,11.0,81.0, 0), v10, z5, tool0;
	MoveL Offs(p0,10.0,81.0, 0), v10, z5, tool0;
	MoveL Offs(p0,11.0,83.0, 0), v10, z5, tool0;
	MoveL Offs(p0,12.0,86.0, 0), v10, z5, tool0;
	MoveL Offs(p0,12.0,86.0, 0), v10, z5, tool0;
	MoveL Offs(p0,12.0,86.0, 0), v10, z5, tool0;
	MoveL Offs(p0,12.0,87.0, 0), v10, z5, tool0;
	MoveL Offs(p0,12.0,87.0, 0), v10, z5, tool0;
	MoveL Offs(p0,12.0,87.0, 0), v10, z5, tool0;
	MoveL Offs(p0,12.0,89.0, 0), v10, z5, tool0;
	MoveL Offs(p0,13.0,90.0, 0), v10, z5, tool0;
	MoveL Offs(p0,13.0,90.0, 0), v10, z5, tool0;
	MoveL Offs(p0,17.0,91.0, 0), v10, z5, tool0;
	MoveL Offs(p0,17.0,91.0, 0), v10, z5, tool0;
	MoveL Offs(p0,18.0,91.0, 0), v10, z5, tool0;
	MoveL Offs(p0,19.0,91.0, 0), v10, z5, tool0;
	MoveL Offs(p0,20.0,91.0, 0), v10, z5, tool0;
	MoveL Offs(p0,20.0,90.0, 0), v10, z5, tool0;
	MoveL Offs(p0,21.0,90.0, 0), v10, z5, tool0;
	MoveL Offs(p0,21.0,90.0, 0), v10, z5, tool0;
	MoveJ Offs(p0,21.0,90.0, 20), v10, z1, tool0;
	MoveJ Offs(p0,84.0,91.0, 20), v10, z1, tool0;
	MoveJ Offs(p0,84.0,91.0, 0), v10, z1, tool0;
	MoveL Offs(p0,84.0,89.0, 0), v10, z5, tool0;
	MoveL Offs(p0,84.0,88.0, 0), v10, z5, tool0;
	MoveL Offs(p0,84.0,88.0, 0), v10, z5, tool0;
	MoveL Offs(p0,82.0,86.0, 0), v10, z5, tool0;
	MoveL Offs(p0,83.0,86.0, 0), v10, z5, tool0;
	MoveL Offs(p0,80.0,84.0, 0), v10, z5, tool0;
	MoveL Offs(p0,77.0,83.0, 0), v10, z5, tool0;
	MoveL Offs(p0,75.0,82.0, 0), v10, z5, tool0;
	MoveL Offs(p0,72.0,81.0, 0), v10, z5, tool0;
	MoveL Offs(p0,70.0,79.0, 0), v10, z5, tool0;
	MoveL Offs(p0,68.0,78.0, 0), v10, z5, tool0;
	MoveL Offs(p0,66.0,77.0, 0), v10, z5, tool0;
	MoveL Offs(p0,64.0,75.0, 0), v10, z5, tool0;
	MoveL Offs(p0,63.0,74.0, 0), v10, z5, tool0;
	MoveL Offs(p0,62.0,73.0, 0), v10, z5, tool0;
	MoveL Offs(p0,60.0,71.0, 0), v10, z5, tool0;
	MoveL Offs(p0,60.0,70.0, 0), v10, z5, tool0;
	MoveL Offs(p0,60.0,70.0, 0), v10, z5, tool0;
	MoveL Offs(p0,60.0,70.0, 0), v10, z5, tool0;
	MoveL Offs(p0,61.0,71.0, 0), v10, z5, tool0;
	MoveL Offs(p0,66.0,75.0, 0), v10, z5, tool0;
	MoveL Offs(p0,67.0,76.0, 0), v10, z5, tool0;
	MoveL Offs(p0,68.0,77.0, 0), v10, z5, tool0;
	MoveL Offs(p0,69.0,78.0, 0), v10, z5, tool0;
	MoveL Offs(p0,70.0,78.0, 0), v10, z5, tool0;
	MoveL Offs(p0,72.0,79.0, 0), v10, z5, tool0;
	MoveL Offs(p0,73.0,80.0, 0), v10, z5, tool0;
	MoveL Offs(p0,75.0,81.0, 0), v10, z5, tool0;
	MoveL Offs(p0,76.0,81.0, 0), v10, z5, tool0;
	MoveL Offs(p0,79.0,82.0, 0), v10, z5, tool0;
	MoveL Offs(p0,81.0,83.0, 0), v10, z5, tool0;
	MoveL Offs(p0,82.0,83.0, 0), v10, z5, tool0;
	MoveL Offs(p0,82.0,83.0, 0), v10, z5, tool0;
	MoveL Offs(p0,83.0,83.0, 0), v10, z5, tool0;
	MoveL Offs(p0,84.0,83.0, 0), v10, z5, tool0;
	MoveL Offs(p0,84.0,83.0, 0), v10, z5, tool0;
	MoveL Offs(p0,85.0,83.0, 0), v10, z5, tool0;
	MoveL Offs(p0,85.0,83.0, 0), v10, z5, tool0;
	MoveL Offs(p0,88.0,83.0, 0), v10, z5, tool0;
	MoveL Offs(p0,88.0,83.0, 0), v10, z5, tool0;
	MoveL Offs(p0,89.0,83.0, 0), v10, z5, tool0;
	MoveL Offs(p0,90.0,83.0, 0), v10, z5, tool0;
	MoveL Offs(p0,92.0,84.0, 0), v10, z5, tool0;
	MoveL Offs(p0,93.0,84.0, 0), v10, z5, tool0;
	MoveL Offs(p0,94.0,84.0, 0), v10, z5, tool0;
	MoveL Offs(p0,95.0,84.0, 0), v10, z5, tool0;
	MoveL Offs(p0,96.0,84.0, 0), v10, z5, tool0;
	MoveL Offs(p0,97.0,84.0, 0), v10, z5, tool0;
	MoveL Offs(p0,97.0,84.0, 0), v10, z5, tool0;
	MoveL Offs(p0,98.0,83.0, 0), v10, z5, tool0;
	MoveL Offs(p0,99.0,83.0, 0), v10, z5, tool0;
	MoveL Offs(p0,100.0,83.0, 0), v10, z5, tool0;
	MoveL Offs(p0,98.0,82.0, 0), v10, z5, tool0;
	MoveL Offs(p0,95.0,79.0, 0), v10, z5, tool0;
	MoveL Offs(p0,94.0,77.0, 0), v10, z5, tool0;
	MoveL Offs(p0,93.0,76.0, 0), v10, z5, tool0;
	MoveL Offs(p0,91.0,74.0, 0), v10, z5, tool0;
	MoveL Offs(p0,90.0,72.0, 0), v10, z5, tool0;
	MoveL Offs(p0,89.0,70.0, 0), v10, z5, tool0;
	MoveL Offs(p0,88.0,68.0, 0), v10, z5, tool0;
	MoveL Offs(p0,87.0,66.0, 0), v10, z5, tool0;
	MoveL Offs(p0,85.0,64.0, 0), v10, z5, tool0;
	MoveL Offs(p0,85.0,64.0, 0), v10, z5, tool0;
	MoveL Offs(p0,82.0,65.0, 0), v10, z5, tool0;
	MoveL Offs(p0,82.0,66.0, 0), v10, z5, tool0;
	MoveL Offs(p0,82.0,66.0, 0), v10, z5, tool0;
	MoveL Offs(p0,81.0,66.0, 0), v10, z5, tool0;
	MoveL Offs(p0,81.0,67.0, 0), v10, z5, tool0;
	MoveL Offs(p0,81.0,67.0, 0), v10, z5, tool0;
	MoveL Offs(p0,79.0,70.0, 0), v10, z5, tool0;
	MoveL Offs(p0,78.0,70.0, 0), v10, z5, tool0;
	MoveL Offs(p0,77.0,71.0, 0), v10, z5, tool0;
	MoveL Offs(p0,75.0,71.0, 0), v10, z5, tool0;
	MoveL Offs(p0,74.0,72.0, 0), v10, z5, tool0;
	MoveL Offs(p0,73.0,72.0, 0), v10, z5, tool0;
	MoveL Offs(p0,72.0,72.0, 0), v10, z5, tool0;
	MoveL Offs(p0,71.0,72.0, 0), v10, z5, tool0;
	MoveL Offs(p0,69.0,71.0, 0), v10, z5, tool0;
	MoveL Offs(p0,68.0,71.0, 0), v10, z5, tool0;
	MoveL Offs(p0,67.0,70.0, 0), v10, z5, tool0;
	MoveL Offs(p0,67.0,70.0, 0), v10, z5, tool0;
	MoveL Offs(p0,66.0,70.0, 0), v10, z5, tool0;
	MoveL Offs(p0,65.0,69.0, 0), v10, z5, tool0;
	MoveL Offs(p0,65.0,69.0, 0), v10, z5, tool0;
	MoveL Offs(p0,64.0,68.0, 0), v10, z5, tool0;
	MoveL Offs(p0,61.0,66.0, 0), v10, z5, tool0;
	MoveL Offs(p0,60.0,66.0, 0), v10, z5, tool0;
	MoveL Offs(p0,59.0,66.0, 0), v10, z5, tool0;
	MoveL Offs(p0,59.0,66.0, 0), v10, z5, tool0;
	MoveL Offs(p0,58.0,66.0, 0), v10, z5, tool0;
	MoveL Offs(p0,58.0,67.0, 0), v10, z5, tool0;
	MoveL Offs(p0,57.0,68.0, 0), v10, z5, tool0;
	MoveL Offs(p0,57.0,68.0, 0), v10, z5, tool0;
	MoveL Offs(p0,55.0,71.0, 0), v10, z5, tool0;
	MoveL Offs(p0,55.0,71.0, 0), v10, z5, tool0;
	MoveL Offs(p0,54.0,72.0, 0), v10, z5, tool0;
	MoveL Offs(p0,53.0,73.0, 0), v10, z5, tool0;
	MoveL Offs(p0,52.0,74.0, 0), v10, z5, tool0;
	MoveL Offs(p0,51.0,74.0, 0), v10, z5, tool0;
	MoveL Offs(p0,50.0,75.0, 0), v10, z5, tool0;
	MoveL Offs(p0,50.0,76.0, 0), v10, z5, tool0;
	MoveL Offs(p0,47.0,77.0, 0), v10, z5, tool0;
	MoveL Offs(p0,46.0,77.0, 0), v10, z5, tool0;
	MoveL Offs(p0,45.0,78.0, 0), v10, z5, tool0;
	MoveL Offs(p0,44.0,78.0, 0), v10, z5, tool0;
	MoveL Offs(p0,44.0,78.0, 0), v10, z5, tool0;
	MoveL Offs(p0,43.0,78.0, 0), v10, z5, tool0;
	MoveL Offs(p0,42.0,78.0, 0), v10, z5, tool0;
	MoveL Offs(p0,42.0,78.0, 0), v10, z5, tool0;
	MoveL Offs(p0,44.0,80.0, 0), v10, z5, tool0;
	MoveL Offs(p0,45.0,81.0, 0), v10, z5, tool0;
	MoveL Offs(p0,48.0,82.0, 0), v10, z5, tool0;
	MoveL Offs(p0,52.0,84.0, 0), v10, z5, tool0;
	MoveL Offs(p0,55.0,85.0, 0), v10, z5, tool0;
	MoveL Offs(p0,59.0,86.0, 0), v10, z5, tool0;
	MoveL Offs(p0,62.0,87.0, 0), v10, z5, tool0;
	MoveL Offs(p0,65.0,88.0, 0), v10, z5, tool0;
	MoveL Offs(p0,68.0,89.0, 0), v10, z5, tool0;
	MoveL Offs(p0,71.0,90.0, 0), v10, z5, tool0;
	MoveL Offs(p0,74.0,91.0, 0), v10, z5, tool0;
	MoveL Offs(p0,77.0,91.0, 0), v10, z5, tool0;
	MoveL Offs(p0,79.0,91.0, 0), v10, z5, tool0;
	MoveL Offs(p0,80.0,91.0, 0), v10, z5, tool0;
	MoveL Offs(p0,81.0,91.0, 0), v10, z5, tool0;
	MoveL Offs(p0,82.0,91.0, 0), v10, z5, tool0;
	MoveL Offs(p0,83.0,91.0, 0), v10, z5, tool0;
	MoveL Offs(p0,83.0,91.0, 0), v10, z5, tool0;
	MoveL Offs(p0,84.0,91.0, 0), v10, z5, tool0;
	MoveL Offs(p0,84.0,91.0, 0), v10, z5, tool0;
	MoveL Offs(p0,84.0,91.0, 0), v10, z5, tool0;
	MoveJ Offs(p0,84.0,91.0, 20), v10, z1, tool0;
	MoveJ Offs(p0,10.0,83.0, 20), v10, z1, tool0;
	MoveJ Offs(p0,10.0,83.0, 0), v10, z1, tool0;
	MoveL Offs(p0,9.0,81.0, 0), v10, z5, tool0;
	MoveL Offs(p0,9.0,80.0, 0), v10, z5, tool0;
	MoveL Offs(p0,9.0,80.0, 0), v10, z5, tool0;
	MoveL Offs(p0,9.0,80.0, 0), v10, z5, tool0;
	MoveL Offs(p0,9.0,80.0, 0), v10, z5, tool0;
	MoveL Offs(p0,9.0,84.0, 0), v10, z5, tool0;
	MoveL Offs(p0,9.0,84.0, 0), v10, z5, tool0;
	MoveL Offs(p0,9.0,84.0, 0), v10, z5, tool0;
	MoveL Offs(p0,9.0,85.0, 0), v10, z5, tool0;
	MoveL Offs(p0,10.0,85.0, 0), v10, z5, tool0;
	MoveL Offs(p0,10.0,86.0, 0), v10, z5, tool0;
	MoveL Offs(p0,11.0,85.0, 0), v10, z5, tool0;
	MoveL Offs(p0,11.0,84.0, 0), v10, z5, tool0;
	MoveL Offs(p0,11.0,84.0, 0), v10, z5, tool0;
	MoveL Offs(p0,11.0,83.0, 0), v10, z5, tool0;
	MoveL Offs(p0,10.0,83.0, 0), v10, z5, tool0;
	MoveL Offs(p0,10.0,83.0, 0), v10, z5, tool0;
	MoveJ Offs(p0,10.0,83.0, 20), v10, z1, tool0;
	MoveJ Offs(p0,100.0,81.0, 20), v10, z1, tool0;
	MoveJ Offs(p0,100.0,81.0, 0), v10, z1, tool0;
	MoveL Offs(p0,99.0,79.0, 0), v10, z5, tool0;
	MoveL Offs(p0,99.0,78.0, 0), v10, z5, tool0;
	MoveL Offs(p0,99.0,78.0, 0), v10, z5, tool0;
	MoveL Offs(p0,98.0,77.0, 0), v10, z5, tool0;
	MoveL Offs(p0,98.0,77.0, 0), v10, z5, tool0;
	MoveL Offs(p0,95.0,75.0, 0), v10, z5, tool0;
	MoveL Offs(p0,95.0,74.0, 0), v10, z5, tool0;
	MoveL Offs(p0,94.0,74.0, 0), v10, z5, tool0;
	MoveL Offs(p0,93.0,73.0, 0), v10, z5, tool0;
	MoveL Offs(p0,93.0,73.0, 0), v10, z5, tool0;
	MoveL Offs(p0,92.0,73.0, 0), v10, z5, tool0;
	MoveL Offs(p0,92.0,73.0, 0), v10, z5, tool0;
	MoveL Offs(p0,94.0,76.0, 0), v10, z5, tool0;
	MoveL Offs(p0,95.0,77.0, 0), v10, z5, tool0;
	MoveL Offs(p0,95.0,77.0, 0), v10, z5, tool0;
	MoveL Offs(p0,96.0,78.0, 0), v10, z5, tool0;
	MoveL Offs(p0,97.0,79.0, 0), v10, z5, tool0;
	MoveL Offs(p0,98.0,80.0, 0), v10, z5, tool0;
	MoveL Offs(p0,100.0,81.0, 0), v10, z5, tool0;
	MoveL Offs(p0,100.0,82.0, 0), v10, z5, tool0;
	MoveL Offs(p0,100.0,82.0, 0), v10, z5, tool0;
	MoveL Offs(p0,100.0,81.0, 0), v10, z5, tool0;
	MoveL Offs(p0,100.0,81.0, 0), v10, z5, tool0;
	MoveL Offs(p0,100.0,81.0, 0), v10, z5, tool0;
	MoveL Offs(p0,100.0,81.0, 0), v10, z5, tool0;
	MoveJ Offs(p0,100.0,81.0, 20), v10, z1, tool0;
	MoveJ Offs(p0,103.0,81.0, 20), v10, z1, tool0;
	MoveJ Offs(p0,103.0,81.0, 0), v10, z1, tool0;
	MoveL Offs(p0,103.0,81.0, 0), v10, z5, tool0;
	MoveJ Offs(p0,103.0,81.0, 20), v10, z1, tool0;
	MoveJ Offs(p0,105.0,80.0, 20), v10, z1, tool0;
	MoveJ Offs(p0,105.0,80.0, 0), v10, z1, tool0;
	MoveL Offs(p0,103.0,76.0, 0), v10, z5, tool0;
	MoveL Offs(p0,102.0,74.0, 0), v10, z5, tool0;
	MoveL Offs(p0,102.0,73.0, 0), v10, z5, tool0;
	MoveL Offs(p0,101.0,71.0, 0), v10, z5, tool0;
	MoveL Offs(p0,101.0,69.0, 0), v10, z5, tool0;
	MoveL Offs(p0,102.0,67.0, 0), v10, z5, tool0;
	MoveL Offs(p0,103.0,65.0, 0), v10, z5, tool0;
	MoveL Offs(p0,104.0,64.0, 0), v10, z5, tool0;
	MoveL Offs(p0,105.0,62.0, 0), v10, z5, tool0;
	MoveL Offs(p0,109.0,59.0, 0), v10, z5, tool0;
	MoveL Offs(p0,110.0,58.0, 0), v10, z5, tool0;
	MoveL Offs(p0,112.0,57.0, 0), v10, z5, tool0;
	MoveL Offs(p0,113.0,55.0, 0), v10, z5, tool0;
	MoveL Offs(p0,115.0,54.0, 0), v10, z5, tool0;
	MoveL Offs(p0,116.0,52.0, 0), v10, z5, tool0;
	MoveL Offs(p0,117.0,50.0, 0), v10, z5, tool0;
	MoveL Offs(p0,118.0,49.0, 0), v10, z5, tool0;
	MoveL Offs(p0,120.0,46.0, 0), v10, z5, tool0;
	MoveL Offs(p0,121.0,44.0, 0), v10, z5, tool0;
	MoveL Offs(p0,122.0,43.0, 0), v10, z5, tool0;
	MoveL Offs(p0,122.0,41.0, 0), v10, z5, tool0;
	MoveL Offs(p0,123.0,39.0, 0), v10, z5, tool0;
	MoveL Offs(p0,123.0,37.0, 0), v10, z5, tool0;
	MoveL Offs(p0,123.0,36.0, 0), v10, z5, tool0;
	MoveL Offs(p0,123.0,34.0, 0), v10, z5, tool0;
	MoveL Offs(p0,124.0,32.0, 0), v10, z5, tool0;
	MoveL Offs(p0,123.0,29.0, 0), v10, z5, tool0;
	MoveL Offs(p0,123.0,28.0, 0), v10, z5, tool0;
	MoveL Offs(p0,123.0,27.0, 0), v10, z5, tool0;
	MoveL Offs(p0,123.0,26.0, 0), v10, z5, tool0;
	MoveL Offs(p0,122.0,25.0, 0), v10, z5, tool0;
	MoveL Offs(p0,122.0,24.0, 0), v10, z5, tool0;
	MoveL Offs(p0,121.0,23.0, 0), v10, z5, tool0;
	MoveL Offs(p0,121.0,22.0, 0), v10, z5, tool0;
	MoveL Offs(p0,119.0,19.0, 0), v10, z5, tool0;
	MoveL Offs(p0,117.0,17.0, 0), v10, z5, tool0;
	MoveL Offs(p0,116.0,16.0, 0), v10, z5, tool0;
	MoveL Offs(p0,114.0,15.0, 0), v10, z5, tool0;
	MoveL Offs(p0,113.0,14.0, 0), v10, z5, tool0;
	MoveL Offs(p0,111.0,14.0, 0), v10, z5, tool0;
	MoveL Offs(p0,109.0,13.0, 0), v10, z5, tool0;
	MoveL Offs(p0,108.0,13.0, 0), v10, z5, tool0;
	MoveL Offs(p0,106.0,14.0, 0), v10, z5, tool0;
	MoveL Offs(p0,104.0,15.0, 0), v10, z5, tool0;
	MoveL Offs(p0,103.0,15.0, 0), v10, z5, tool0;
	MoveL Offs(p0,103.0,16.0, 0), v10, z5, tool0;
	MoveL Offs(p0,102.0,16.0, 0), v10, z5, tool0;
	MoveL Offs(p0,102.0,17.0, 0), v10, z5, tool0;
	MoveL Offs(p0,102.0,18.0, 0), v10, z5, tool0;
	MoveL Offs(p0,101.0,18.0, 0), v10, z5, tool0;
	MoveL Offs(p0,101.0,19.0, 0), v10, z5, tool0;
	MoveL Offs(p0,103.0,17.0, 0), v10, z5, tool0;
	MoveL Offs(p0,103.0,16.0, 0), v10, z5, tool0;
	MoveL Offs(p0,104.0,16.0, 0), v10, z5, tool0;
	MoveL Offs(p0,104.0,15.0, 0), v10, z5, tool0;
	MoveL Offs(p0,105.0,15.0, 0), v10, z5, tool0;
	MoveL Offs(p0,105.0,15.0, 0), v10, z5, tool0;
	MoveL Offs(p0,105.0,15.0, 0), v10, z5, tool0;
	MoveL Offs(p0,109.0,15.0, 0), v10, z5, tool0;
	MoveL Offs(p0,109.0,15.0, 0), v10, z5, tool0;
	MoveL Offs(p0,110.0,15.0, 0), v10, z5, tool0;
	MoveL Offs(p0,111.0,15.0, 0), v10, z5, tool0;
	MoveL Offs(p0,112.0,16.0, 0), v10, z5, tool0;
	MoveL Offs(p0,113.0,16.0, 0), v10, z5, tool0;
	MoveL Offs(p0,115.0,18.0, 0), v10, z5, tool0;
	MoveL Offs(p0,116.0,19.0, 0), v10, z5, tool0;
	MoveL Offs(p0,117.0,20.0, 0), v10, z5, tool0;
	MoveL Offs(p0,118.0,21.0, 0), v10, z5, tool0;
	MoveL Offs(p0,119.0,23.0, 0), v10, z5, tool0;
	MoveL Offs(p0,120.0,24.0, 0), v10, z5, tool0;
	MoveL Offs(p0,120.0,26.0, 0), v10, z5, tool0;
	MoveL Offs(p0,121.0,27.0, 0), v10, z5, tool0;
	MoveL Offs(p0,121.0,29.0, 0), v10, z5, tool0;
	MoveL Offs(p0,121.0,32.0, 0), v10, z5, tool0;
	MoveL Offs(p0,121.0,35.0, 0), v10, z5, tool0;
	MoveL Offs(p0,121.0,37.0, 0), v10, z5, tool0;
	MoveL Offs(p0,120.0,40.0, 0), v10, z5, tool0;
	MoveL Offs(p0,119.0,43.0, 0), v10, z5, tool0;
	MoveL Offs(p0,118.0,46.0, 0), v10, z5, tool0;
	MoveL Offs(p0,116.0,48.0, 0), v10, z5, tool0;
	MoveL Offs(p0,114.0,51.0, 0), v10, z5, tool0;
	MoveL Offs(p0,112.0,53.0, 0), v10, z5, tool0;
	MoveL Offs(p0,110.0,55.0, 0), v10, z5, tool0;
	MoveL Offs(p0,108.0,57.0, 0), v10, z5, tool0;
	MoveL Offs(p0,108.0,57.0, 0), v10, z5, tool0;
	MoveL Offs(p0,108.0,57.0, 0), v10, z5, tool0;
	MoveL Offs(p0,107.0,57.0, 0), v10, z5, tool0;
	MoveL Offs(p0,107.0,57.0, 0), v10, z5, tool0;
	MoveL Offs(p0,105.0,59.0, 0), v10, z5, tool0;
	MoveL Offs(p0,105.0,59.0, 0), v10, z5, tool0;
	MoveL Offs(p0,103.0,61.0, 0), v10, z5, tool0;
	MoveL Offs(p0,102.0,62.0, 0), v10, z5, tool0;
	MoveL Offs(p0,101.0,63.0, 0), v10, z5, tool0;
	MoveL Offs(p0,101.0,64.0, 0), v10, z5, tool0;
	MoveL Offs(p0,100.0,65.0, 0), v10, z5, tool0;
	MoveL Offs(p0,100.0,66.0, 0), v10, z5, tool0;
	MoveL Offs(p0,99.0,68.0, 0), v10, z5, tool0;
	MoveL Offs(p0,99.0,69.0, 0), v10, z5, tool0;
	MoveL Offs(p0,99.0,71.0, 0), v10, z5, tool0;
	MoveL Offs(p0,99.0,73.0, 0), v10, z5, tool0;
	MoveL Offs(p0,99.0,74.0, 0), v10, z5, tool0;
	MoveL Offs(p0,100.0,75.0, 0), v10, z5, tool0;
	MoveL Offs(p0,100.0,76.0, 0), v10, z5, tool0;
	MoveL Offs(p0,100.0,77.0, 0), v10, z5, tool0;
	MoveL Offs(p0,101.0,78.0, 0), v10, z5, tool0;
	MoveL Offs(p0,101.0,78.0, 0), v10, z5, tool0;
	MoveL Offs(p0,102.0,79.0, 0), v10, z5, tool0;
	MoveL Offs(p0,103.0,80.0, 0), v10, z5, tool0;
	MoveL Offs(p0,105.0,80.0, 0), v10, z5, tool0;
	MoveL Offs(p0,105.0,80.0, 0), v10, z5, tool0;
	MoveL Offs(p0,105.0,80.0, 0), v10, z5, tool0;
	MoveJ Offs(p0,105.0,80.0, 20), v10, z1, tool0;
	MoveJ Offs(p0,15.0,79.0, 20), v10, z1, tool0;
	MoveJ Offs(p0,15.0,79.0, 0), v10, z1, tool0;
	MoveL Offs(p0,17.0,78.0, 0), v10, z5, tool0;
	MoveL Offs(p0,17.0,78.0, 0), v10, z5, tool0;
	MoveL Offs(p0,17.0,78.0, 0), v10, z5, tool0;
	MoveL Offs(p0,18.0,77.0, 0), v10, z5, tool0;
	MoveL Offs(p0,16.0,75.0, 0), v10, z5, tool0;
	MoveL Offs(p0,15.0,72.0, 0), v10, z5, tool0;
	MoveL Offs(p0,14.0,72.0, 0), v10, z5, tool0;
	MoveL Offs(p0,14.0,72.0, 0), v10, z5, tool0;
	MoveL Offs(p0,14.0,71.0, 0), v10, z5, tool0;
	MoveL Offs(p0,14.0,71.0, 0), v10, z5, tool0;
	MoveL Offs(p0,13.0,70.0, 0), v10, z5, tool0;
	MoveL Offs(p0,12.0,68.0, 0), v10, z5, tool0;
	MoveL Offs(p0,12.0,68.0, 0), v10, z5, tool0;
	MoveL Offs(p0,12.0,68.0, 0), v10, z5, tool0;
	MoveL Offs(p0,11.0,68.0, 0), v10, z5, tool0;
	MoveL Offs(p0,11.0,68.0, 0), v10, z5, tool0;
	MoveL Offs(p0,10.0,67.0, 0), v10, z5, tool0;
	MoveL Offs(p0,8.0,67.0, 0), v10, z5, tool0;
	MoveL Offs(p0,8.0,67.0, 0), v10, z5, tool0;
	MoveL Offs(p0,8.0,67.0, 0), v10, z5, tool0;
	MoveL Offs(p0,7.0,70.0, 0), v10, z5, tool0;
	MoveL Offs(p0,7.0,71.0, 0), v10, z5, tool0;
	MoveL Offs(p0,7.0,72.0, 0), v10, z5, tool0;
	MoveL Offs(p0,7.0,74.0, 0), v10, z5, tool0;
	MoveL Offs(p0,7.0,75.0, 0), v10, z5, tool0;
	MoveL Offs(p0,7.0,76.0, 0), v10, z5, tool0;
	MoveL Offs(p0,7.0,76.0, 0), v10, z5, tool0;
	MoveL Offs(p0,7.0,77.0, 0), v10, z5, tool0;
	MoveL Offs(p0,7.0,77.0, 0), v10, z5, tool0;
	MoveL Offs(p0,7.0,77.0, 0), v10, z5, tool0;
	MoveL Offs(p0,7.0,78.0, 0), v10, z5, tool0;
	MoveL Offs(p0,8.0,78.0, 0), v10, z5, tool0;
	MoveL Offs(p0,10.0,79.0, 0), v10, z5, tool0;
	MoveL Offs(p0,11.0,79.0, 0), v10, z5, tool0;
	MoveL Offs(p0,11.0,80.0, 0), v10, z5, tool0;
	MoveL Offs(p0,12.0,80.0, 0), v10, z5, tool0;
	MoveL Offs(p0,13.0,79.0, 0), v10, z5, tool0;
	MoveL Offs(p0,14.0,79.0, 0), v10, z5, tool0;
	MoveL Offs(p0,15.0,79.0, 0), v10, z5, tool0;
	MoveL Offs(p0,15.0,79.0, 0), v10, z5, tool0;
	MoveJ Offs(p0,15.0,79.0, 20), v10, z1, tool0;
	MoveJ Offs(p0,6.0,71.0, 20), v10, z1, tool0;
	MoveJ Offs(p0,6.0,71.0, 0), v10, z1, tool0;
	MoveL Offs(p0,6.0,66.0, 0), v10, z5, tool0;
	MoveL Offs(p0,5.0,65.0, 0), v10, z5, tool0;
	MoveL Offs(p0,3.0,64.0, 0), v10, z5, tool0;
	MoveL Offs(p0,3.0,65.0, 0), v10, z5, tool0;
	MoveL Offs(p0,3.0,67.0, 0), v10, z5, tool0;
	MoveL Offs(p0,3.0,67.0, 0), v10, z5, tool0;
	MoveL Offs(p0,3.0,68.0, 0), v10, z5, tool0;
	MoveL Offs(p0,3.0,68.0, 0), v10, z5, tool0;
	MoveL Offs(p0,3.0,69.0, 0), v10, z5, tool0;
	MoveL Offs(p0,4.0,72.0, 0), v10, z5, tool0;
	MoveL Offs(p0,4.0,73.0, 0), v10, z5, tool0;
	MoveL Offs(p0,5.0,73.0, 0), v10, z5, tool0;
	MoveL Offs(p0,5.0,74.0, 0), v10, z5, tool0;
	MoveL Offs(p0,5.0,75.0, 0), v10, z5, tool0;
	MoveL Offs(p0,6.0,76.0, 0), v10, z5, tool0;
	MoveL Offs(p0,6.0,76.0, 0), v10, z5, tool0;
	MoveL Offs(p0,6.0,76.0, 0), v10, z5, tool0;
	MoveL Offs(p0,6.0,73.0, 0), v10, z5, tool0;
	MoveL Offs(p0,6.0,73.0, 0), v10, z5, tool0;
	MoveL Offs(p0,6.0,72.0, 0), v10, z5, tool0;
	MoveL Offs(p0,6.0,71.0, 0), v10, z5, tool0;
	MoveL Offs(p0,6.0,71.0, 0), v10, z5, tool0;
	MoveJ Offs(p0,6.0,71.0, 20), v10, z1, tool0;
	MoveJ Offs(p0,19.0,75.0, 20), v10, z1, tool0;
	MoveJ Offs(p0,19.0,75.0, 0), v10, z1, tool0;
	MoveL Offs(p0,18.0,72.0, 0), v10, z5, tool0;
	MoveL Offs(p0,18.0,72.0, 0), v10, z5, tool0;
	MoveL Offs(p0,18.0,71.0, 0), v10, z5, tool0;
	MoveL Offs(p0,18.0,71.0, 0), v10, z5, tool0;
	MoveL Offs(p0,17.0,70.0, 0), v10, z5, tool0;
	MoveL Offs(p0,17.0,70.0, 0), v10, z5, tool0;
	MoveL Offs(p0,17.0,69.0, 0), v10, z5, tool0;
	MoveL Offs(p0,15.0,67.0, 0), v10, z5, tool0;
	MoveL Offs(p0,15.0,66.0, 0), v10, z5, tool0;
	MoveL Offs(p0,15.0,66.0, 0), v10, z5, tool0;
	MoveL Offs(p0,15.0,66.0, 0), v10, z5, tool0;
	MoveL Offs(p0,15.0,67.0, 0), v10, z5, tool0;
	MoveL Offs(p0,19.0,70.0, 0), v10, z5, tool0;
	MoveL Offs(p0,19.0,70.0, 0), v10, z5, tool0;
	MoveL Offs(p0,19.0,70.0, 0), v10, z5, tool0;
	MoveL Offs(p0,19.0,69.0, 0), v10, z5, tool0;
	MoveL Offs(p0,19.0,69.0, 0), v10, z5, tool0;
	MoveL Offs(p0,19.0,69.0, 0), v10, z5, tool0;
	MoveL Offs(p0,18.0,67.0, 0), v10, z5, tool0;
	MoveL Offs(p0,18.0,66.0, 0), v10, z5, tool0;
	MoveL Offs(p0,17.0,65.0, 0), v10, z5, tool0;
	MoveL Offs(p0,17.0,64.0, 0), v10, z5, tool0;
	MoveL Offs(p0,16.0,63.0, 0), v10, z5, tool0;
	MoveL Offs(p0,16.0,62.0, 0), v10, z5, tool0;
	MoveL Offs(p0,15.0,61.0, 0), v10, z5, tool0;
	MoveL Offs(p0,15.0,61.0, 0), v10, z5, tool0;
	MoveL Offs(p0,17.0,58.0, 0), v10, z5, tool0;
	MoveL Offs(p0,16.0,57.0, 0), v10, z5, tool0;
	MoveL Offs(p0,15.0,57.0, 0), v10, z5, tool0;
	MoveL Offs(p0,15.0,56.0, 0), v10, z5, tool0;
	MoveL Offs(p0,14.0,55.0, 0), v10, z5, tool0;
	MoveL Offs(p0,14.0,55.0, 0), v10, z5, tool0;
	MoveL Offs(p0,13.0,55.0, 0), v10, z5, tool0;
	MoveL Offs(p0,12.0,57.0, 0), v10, z5, tool0;
	MoveL Offs(p0,12.0,58.0, 0), v10, z5, tool0;
	MoveL Offs(p0,12.0,59.0, 0), v10, z5, tool0;
	MoveL Offs(p0,12.0,60.0, 0), v10, z5, tool0;
	MoveL Offs(p0,12.0,61.0, 0), v10, z5, tool0;
	MoveL Offs(p0,12.0,63.0, 0), v10, z5, tool0;
	MoveL Offs(p0,12.0,64.0, 0), v10, z5, tool0;
	MoveL Offs(p0,12.0,65.0, 0), v10, z5, tool0;
	MoveL Offs(p0,12.0,65.0, 0), v10, z5, tool0;
	MoveL Offs(p0,12.0,66.0, 0), v10, z5, tool0;
	MoveL Offs(p0,13.0,66.0, 0), v10, z5, tool0;
	MoveL Offs(p0,13.0,67.0, 0), v10, z5, tool0;
	MoveL Offs(p0,13.0,68.0, 0), v10, z5, tool0;
	MoveL Offs(p0,15.0,70.0, 0), v10, z5, tool0;
	MoveL Offs(p0,15.0,71.0, 0), v10, z5, tool0;
	MoveL Offs(p0,16.0,72.0, 0), v10, z5, tool0;
	MoveL Offs(p0,16.0,73.0, 0), v10, z5, tool0;
	MoveL Offs(p0,17.0,74.0, 0), v10, z5, tool0;
	MoveL Offs(p0,17.0,75.0, 0), v10, z5, tool0;
	MoveL Offs(p0,18.0,75.0, 0), v10, z5, tool0;
	MoveL Offs(p0,18.0,75.0, 0), v10, z5, tool0;
	MoveL Offs(p0,18.0,76.0, 0), v10, z5, tool0;
	MoveL Offs(p0,19.0,75.0, 0), v10, z5, tool0;
	MoveJ Offs(p0,19.0,75.0, 20), v10, z1, tool0;
	MoveJ Offs(p0,98.0,73.0, 20), v10, z1, tool0;
	MoveJ Offs(p0,98.0,73.0, 0), v10, z1, tool0;
	MoveL Offs(p0,98.0,71.0, 0), v10, z5, tool0;
	MoveL Offs(p0,98.0,69.0, 0), v10, z5, tool0;
	MoveL Offs(p0,98.0,68.0, 0), v10, z5, tool0;
	MoveL Offs(p0,98.0,66.0, 0), v10, z5, tool0;
	MoveL Offs(p0,99.0,65.0, 0), v10, z5, tool0;
	MoveL Offs(p0,99.0,64.0, 0), v10, z5, tool0;
	MoveL Offs(p0,100.0,62.0, 0), v10, z5, tool0;
	MoveL Offs(p0,101.0,61.0, 0), v10, z5, tool0;
	MoveL Offs(p0,102.0,60.0, 0), v10, z5, tool0;
	MoveL Offs(p0,103.0,59.0, 0), v10, z5, tool0;
	MoveL Offs(p0,101.0,57.0, 0), v10, z5, tool0;
	MoveL Offs(p0,99.0,55.0, 0), v10, z5, tool0;
	MoveL Offs(p0,97.0,54.0, 0), v10, z5, tool0;
	MoveL Offs(p0,96.0,53.0, 0), v10, z5, tool0;
	MoveL Offs(p0,94.0,53.0, 0), v10, z5, tool0;
	MoveL Offs(p0,93.0,52.0, 0), v10, z5, tool0;
	MoveL Offs(p0,91.0,52.0, 0), v10, z5, tool0;
	MoveL Offs(p0,89.0,52.0, 0), v10, z5, tool0;
	MoveL Offs(p0,87.0,52.0, 0), v10, z5, tool0;
	MoveL Offs(p0,86.0,52.0, 0), v10, z5, tool0;
	MoveL Offs(p0,84.0,52.0, 0), v10, z5, tool0;
	MoveL Offs(p0,83.0,52.0, 0), v10, z5, tool0;
	MoveL Offs(p0,82.0,52.0, 0), v10, z5, tool0;
	MoveL Offs(p0,81.0,53.0, 0), v10, z5, tool0;
	MoveL Offs(p0,80.0,53.0, 0), v10, z5, tool0;
	MoveL Offs(p0,80.0,53.0, 0), v10, z5, tool0;
	MoveL Offs(p0,79.0,54.0, 0), v10, z5, tool0;
	MoveL Offs(p0,79.0,54.0, 0), v10, z5, tool0;
	MoveL Offs(p0,78.0,55.0, 0), v10, z5, tool0;
	MoveL Offs(p0,76.0,58.0, 0), v10, z5, tool0;
	MoveL Offs(p0,76.0,58.0, 0), v10, z5, tool0;
	MoveL Offs(p0,76.0,59.0, 0), v10, z5, tool0;
	MoveL Offs(p0,76.0,60.0, 0), v10, z5, tool0;
	MoveL Offs(p0,76.0,60.0, 0), v10, z5, tool0;
	MoveL Offs(p0,75.0,61.0, 0), v10, z5, tool0;
	MoveL Offs(p0,75.0,62.0, 0), v10, z5, tool0;
	MoveL Offs(p0,76.0,65.0, 0), v10, z5, tool0;
	MoveL Offs(p0,76.0,66.0, 0), v10, z5, tool0;
	MoveL Offs(p0,76.0,66.0, 0), v10, z5, tool0;
	MoveL Offs(p0,77.0,67.0, 0), v10, z5, tool0;
	MoveL Offs(p0,77.0,68.0, 0), v10, z5, tool0;
	MoveL Offs(p0,77.0,69.0, 0), v10, z5, tool0;
	MoveL Offs(p0,78.0,69.0, 0), v10, z5, tool0;
	MoveL Offs(p0,78.0,69.0, 0), v10, z5, tool0;
	MoveL Offs(p0,81.0,65.0, 0), v10, z5, tool0;
	MoveL Offs(p0,81.0,64.0, 0), v10, z5, tool0;
	MoveL Offs(p0,82.0,64.0, 0), v10, z5, tool0;
	MoveL Offs(p0,82.0,64.0, 0), v10, z5, tool0;
	MoveL Offs(p0,83.0,64.0, 0), v10, z5, tool0;
	MoveL Offs(p0,84.0,64.0, 0), v10, z5, tool0;
	MoveL Offs(p0,84.0,64.0, 0), v10, z5, tool0;
	MoveL Offs(p0,86.0,64.0, 0), v10, z5, tool0;
	MoveL Offs(p0,87.0,65.0, 0), v10, z5, tool0;
	MoveL Offs(p0,87.0,65.0, 0), v10, z5, tool0;
	MoveL Offs(p0,88.0,66.0, 0), v10, z5, tool0;
	MoveL Offs(p0,88.0,67.0, 0), v10, z5, tool0;
	MoveL Offs(p0,89.0,68.0, 0), v10, z5, tool0;
	MoveL Offs(p0,90.0,70.0, 0), v10, z5, tool0;
	MoveL Offs(p0,91.0,71.0, 0), v10, z5, tool0;
	MoveL Offs(p0,91.0,71.0, 0), v10, z5, tool0;
	MoveL Offs(p0,91.0,71.0, 0), v10, z5, tool0;
	MoveL Offs(p0,92.0,72.0, 0), v10, z5, tool0;
	MoveL Offs(p0,92.0,72.0, 0), v10, z5, tool0;
	MoveL Offs(p0,93.0,72.0, 0), v10, z5, tool0;
	MoveL Offs(p0,93.0,73.0, 0), v10, z5, tool0;
	MoveL Offs(p0,95.0,74.0, 0), v10, z5, tool0;
	MoveL Offs(p0,96.0,74.0, 0), v10, z5, tool0;
	MoveL Offs(p0,96.0,74.0, 0), v10, z5, tool0;
	MoveL Offs(p0,97.0,74.0, 0), v10, z5, tool0;
	MoveL Offs(p0,97.0,74.0, 0), v10, z5, tool0;
	MoveL Offs(p0,97.0,75.0, 0), v10, z5, tool0;
	MoveL Offs(p0,98.0,73.0, 0), v10, z5, tool0;
	MoveL Offs(p0,98.0,73.0, 0), v10, z5, tool0;
	MoveJ Offs(p0,98.0,73.0, 20), v10, z1, tool0;
	MoveJ Offs(p0,105.0,73.0, 20), v10, z1, tool0;
	MoveJ Offs(p0,105.0,73.0, 0), v10, z1, tool0;
	MoveL Offs(p0,105.0,70.0, 0), v10, z5, tool0;
	MoveL Offs(p0,105.0,69.0, 0), v10, z5, tool0;
	MoveL Offs(p0,105.0,68.0, 0), v10, z5, tool0;
	MoveL Offs(p0,105.0,67.0, 0), v10, z5, tool0;
	MoveL Offs(p0,105.0,66.0, 0), v10, z5, tool0;
	MoveL Offs(p0,105.0,65.0, 0), v10, z5, tool0;
	MoveL Offs(p0,105.0,64.0, 0), v10, z5, tool0;
	MoveL Offs(p0,105.0,64.0, 0), v10, z5, tool0;
	MoveL Offs(p0,103.0,66.0, 0), v10, z5, tool0;
	MoveL Offs(p0,103.0,67.0, 0), v10, z5, tool0;
	MoveL Offs(p0,103.0,68.0, 0), v10, z5, tool0;
	MoveL Offs(p0,103.0,70.0, 0), v10, z5, tool0;
	MoveL Offs(p0,103.0,71.0, 0), v10, z5, tool0;
	MoveL Offs(p0,103.0,72.0, 0), v10, z5, tool0;
	MoveL Offs(p0,103.0,72.0, 0), v10, z5, tool0;
	MoveL Offs(p0,103.0,73.0, 0), v10, z5, tool0;
	MoveL Offs(p0,103.0,74.0, 0), v10, z5, tool0;
	MoveL Offs(p0,103.0,74.0, 0), v10, z5, tool0;
	MoveL Offs(p0,105.0,73.0, 0), v10, z5, tool0;
	MoveJ Offs(p0,105.0,73.0, 20), v10, z1, tool0;
	MoveJ Offs(p0,19.0,71.0, 20), v10, z1, tool0;
	MoveJ Offs(p0,19.0,71.0, 0), v10, z1, tool0;
	MoveL Offs(p0,19.0,71.0, 0), v10, z5, tool0;
	MoveJ Offs(p0,19.0,71.0, 20), v10, z1, tool0;
	MoveJ Offs(p0,70.0,68.0, 20), v10, z1, tool0;
	MoveJ Offs(p0,70.0,68.0, 0), v10, z1, tool0;
	MoveL Offs(p0,71.0,66.0, 0), v10, z5, tool0;
	MoveL Offs(p0,71.0,65.0, 0), v10, z5, tool0;
	MoveL Offs(p0,71.0,65.0, 0), v10, z5, tool0;
	MoveL Offs(p0,71.0,64.0, 0), v10, z5, tool0;
	MoveL Offs(p0,71.0,64.0, 0), v10, z5, tool0;
	MoveL Offs(p0,71.0,63.0, 0), v10, z5, tool0;
	MoveL Offs(p0,71.0,61.0, 0), v10, z5, tool0;
	MoveL Offs(p0,71.0,60.0, 0), v10, z5, tool0;
	MoveL Offs(p0,71.0,60.0, 0), v10, z5, tool0;
	MoveL Offs(p0,71.0,60.0, 0), v10, z5, tool0;
	MoveL Offs(p0,71.0,60.0, 0), v10, z5, tool0;
	MoveL Offs(p0,70.0,60.0, 0), v10, z5, tool0;
	MoveL Offs(p0,70.0,60.0, 0), v10, z5, tool0;
	MoveL Offs(p0,67.0,63.0, 0), v10, z5, tool0;
	MoveL Offs(p0,67.0,64.0, 0), v10, z5, tool0;
	MoveL Offs(p0,66.0,65.0, 0), v10, z5, tool0;
	MoveL Offs(p0,66.0,66.0, 0), v10, z5, tool0;
	MoveL Offs(p0,66.0,67.0, 0), v10, z5, tool0;
	MoveL Offs(p0,66.0,68.0, 0), v10, z5, tool0;
	MoveL Offs(p0,66.0,69.0, 0), v10, z5, tool0;
	MoveL Offs(p0,68.0,70.0, 0), v10, z5, tool0;
	MoveL Offs(p0,69.0,70.0, 0), v10, z5, tool0;
	MoveL Offs(p0,69.0,70.0, 0), v10, z5, tool0;
	MoveL Offs(p0,70.0,71.0, 0), v10, z5, tool0;
	MoveL Offs(p0,70.0,71.0, 0), v10, z5, tool0;
	MoveL Offs(p0,70.0,71.0, 0), v10, z5, tool0;
	MoveL Offs(p0,71.0,69.0, 0), v10, z5, tool0;
	MoveL Offs(p0,70.0,68.0, 0), v10, z5, tool0;
	MoveL Offs(p0,70.0,68.0, 0), v10, z5, tool0;
	MoveJ Offs(p0,70.0,68.0, 20), v10, z1, tool0;
	MoveJ Offs(p0,75.0,70.0, 20), v10, z1, tool0;
	MoveJ Offs(p0,75.0,70.0, 0), v10, z1, tool0;
	MoveL Offs(p0,76.0,67.0, 0), v10, z5, tool0;
	MoveL Offs(p0,75.0,65.0, 0), v10, z5, tool0;
	MoveL Offs(p0,75.0,64.0, 0), v10, z5, tool0;
	MoveL Offs(p0,74.0,62.0, 0), v10, z5, tool0;
	MoveL Offs(p0,75.0,61.0, 0), v10, z5, tool0;
	MoveL Offs(p0,75.0,60.0, 0), v10, z5, tool0;
	MoveL Offs(p0,75.0,59.0, 0), v10, z5, tool0;
	MoveL Offs(p0,75.0,58.0, 0), v10, z5, tool0;
	MoveL Offs(p0,76.0,57.0, 0), v10, z5, tool0;
	MoveL Offs(p0,76.0,56.0, 0), v10, z5, tool0;
	MoveL Offs(p0,75.0,55.0, 0), v10, z5, tool0;
	MoveL Offs(p0,74.0,56.0, 0), v10, z5, tool0;
	MoveL Offs(p0,74.0,56.0, 0), v10, z5, tool0;
	MoveL Offs(p0,73.0,56.0, 0), v10, z5, tool0;
	MoveL Offs(p0,71.0,58.0, 0), v10, z5, tool0;
	MoveL Offs(p0,70.0,59.0, 0), v10, z5, tool0;
	MoveL Offs(p0,69.0,59.0, 0), v10, z5, tool0;
	MoveL Offs(p0,69.0,60.0, 0), v10, z5, tool0;
	MoveL Offs(p0,69.0,60.0, 0), v10, z5, tool0;
	MoveL Offs(p0,69.0,60.0, 0), v10, z5, tool0;
	MoveL Offs(p0,69.0,60.0, 0), v10, z5, tool0;
	MoveL Offs(p0,69.0,60.0, 0), v10, z5, tool0;
	MoveL Offs(p0,72.0,62.0, 0), v10, z5, tool0;
	MoveL Offs(p0,72.0,63.0, 0), v10, z5, tool0;
	MoveL Offs(p0,71.0,65.0, 0), v10, z5, tool0;
	MoveL Offs(p0,71.0,66.0, 0), v10, z5, tool0;
	MoveL Offs(p0,71.0,66.0, 0), v10, z5, tool0;
	MoveL Offs(p0,71.0,67.0, 0), v10, z5, tool0;
	MoveL Offs(p0,71.0,68.0, 0), v10, z5, tool0;
	MoveL Offs(p0,71.0,68.0, 0), v10, z5, tool0;
	MoveL Offs(p0,71.0,69.0, 0), v10, z5, tool0;
	MoveL Offs(p0,71.0,69.0, 0), v10, z5, tool0;
	MoveL Offs(p0,74.0,70.0, 0), v10, z5, tool0;
	MoveL Offs(p0,74.0,70.0, 0), v10, z5, tool0;
	MoveL Offs(p0,75.0,70.0, 0), v10, z5, tool0;
	MoveL Offs(p0,75.0,70.0, 0), v10, z5, tool0;
	MoveJ Offs(p0,75.0,70.0, 20), v10, z1, tool0;
	MoveJ Offs(p0,66.0,66.0, 20), v10, z1, tool0;
	MoveJ Offs(p0,66.0,66.0, 0), v10, z1, tool0;
	MoveL Offs(p0,66.0,66.0, 0), v10, z5, tool0;
	MoveJ Offs(p0,66.0,66.0, 20), v10, z1, tool0;
	MoveJ Offs(p0,11.0,66.0, 20), v10, z1, tool0;
	MoveJ Offs(p0,11.0,66.0, 0), v10, z1, tool0;
	MoveL Offs(p0,11.0,63.0, 0), v10, z5, tool0;
	MoveL Offs(p0,11.0,62.0, 0), v10, z5, tool0;
	MoveL Offs(p0,11.0,61.0, 0), v10, z5, tool0;
	MoveL Offs(p0,11.0,60.0, 0), v10, z5, tool0;
	MoveL Offs(p0,11.0,59.0, 0), v10, z5, tool0;
	MoveL Offs(p0,11.0,58.0, 0), v10, z5, tool0;
	MoveL Offs(p0,11.0,57.0, 0), v10, z5, tool0;
	MoveL Offs(p0,11.0,57.0, 0), v10, z5, tool0;
	MoveL Offs(p0,11.0,55.0, 0), v10, z5, tool0;
	MoveL Offs(p0,7.0,53.0, 0), v10, z5, tool0;
	MoveL Offs(p0,7.0,53.0, 0), v10, z5, tool0;
	MoveL Offs(p0,7.0,53.0, 0), v10, z5, tool0;
	MoveL Offs(p0,6.0,55.0, 0), v10, z5, tool0;
	MoveL Offs(p0,6.0,55.0, 0), v10, z5, tool0;
	MoveL Offs(p0,5.0,58.0, 0), v10, z5, tool0;
	MoveL Offs(p0,5.0,59.0, 0), v10, z5, tool0;
	MoveL Offs(p0,5.0,59.0, 0), v10, z5, tool0;
	MoveL Offs(p0,5.0,59.0, 0), v10, z5, tool0;
	MoveL Offs(p0,4.0,60.0, 0), v10, z5, tool0;
	MoveL Offs(p0,4.0,60.0, 0), v10, z5, tool0;
	MoveL Offs(p0,4.0,60.0, 0), v10, z5, tool0;
	MoveL Offs(p0,3.0,60.0, 0), v10, z5, tool0;
	MoveL Offs(p0,2.0,57.0, 0), v10, z5, tool0;
	MoveL Offs(p0,2.0,55.0, 0), v10, z5, tool0;
	MoveL Offs(p0,2.0,54.0, 0), v10, z5, tool0;
	MoveL Offs(p0,2.0,53.0, 0), v10, z5, tool0;
	MoveL Offs(p0,2.0,52.0, 0), v10, z5, tool0;
	MoveL Offs(p0,2.0,51.0, 0), v10, z5, tool0;
	MoveL Offs(p0,2.0,50.0, 0), v10, z5, tool0;
	MoveL Offs(p0,2.0,49.0, 0), v10, z5, tool0;
	MoveL Offs(p0,2.0,48.0, 0), v10, z5, tool0;
	MoveL Offs(p0,1.0,50.0, 0), v10, z5, tool0;
	MoveL Offs(p0,1.0,50.0, 0), v10, z5, tool0;
	MoveL Offs(p0,1.0,51.0, 0), v10, z5, tool0;
	MoveL Offs(p0,1.0,52.0, 0), v10, z5, tool0;
	MoveL Offs(p0,1.0,53.0, 0), v10, z5, tool0;
	MoveL Offs(p0,1.0,56.0, 0), v10, z5, tool0;
	MoveL Offs(p0,2.0,57.0, 0), v10, z5, tool0;
	MoveL Offs(p0,2.0,58.0, 0), v10, z5, tool0;
	MoveL Offs(p0,2.0,59.0, 0), v10, z5, tool0;
	MoveL Offs(p0,2.0,60.0, 0), v10, z5, tool0;
	MoveL Offs(p0,3.0,61.0, 0), v10, z5, tool0;
	MoveL Offs(p0,3.0,61.0, 0), v10, z5, tool0;
	MoveL Offs(p0,4.0,62.0, 0), v10, z5, tool0;
	MoveL Offs(p0,4.0,63.0, 0), v10, z5, tool0;
	MoveL Offs(p0,6.0,65.0, 0), v10, z5, tool0;
	MoveL Offs(p0,7.0,65.0, 0), v10, z5, tool0;
	MoveL Offs(p0,8.0,66.0, 0), v10, z5, tool0;
	MoveL Offs(p0,9.0,66.0, 0), v10, z5, tool0;
	MoveL Offs(p0,9.0,66.0, 0), v10, z5, tool0;
	MoveL Offs(p0,10.0,66.0, 0), v10, z5, tool0;
	MoveL Offs(p0,11.0,66.0, 0), v10, z5, tool0;
	MoveL Offs(p0,11.0,66.0, 0), v10, z5, tool0;
	MoveJ Offs(p0,11.0,66.0, 20), v10, z1, tool0;
	MoveJ Offs(p0,31.0,63.0, 20), v10, z1, tool0;
	MoveJ Offs(p0,31.0,63.0, 0), v10, z1, tool0;
	MoveL Offs(p0,31.0,61.0, 0), v10, z5, tool0;
	MoveL Offs(p0,31.0,59.0, 0), v10, z5, tool0;
	MoveL Offs(p0,30.0,57.0, 0), v10, z5, tool0;
	MoveL Offs(p0,30.0,55.0, 0), v10, z5, tool0;
	MoveL Offs(p0,30.0,53.0, 0), v10, z5, tool0;
	MoveL Offs(p0,29.0,51.0, 0), v10, z5, tool0;
	MoveL Offs(p0,29.0,49.0, 0), v10, z5, tool0;
	MoveL Offs(p0,29.0,47.0, 0), v10, z5, tool0;
	MoveL Offs(p0,28.0,46.0, 0), v10, z5, tool0;
	MoveL Offs(p0,31.0,50.0, 0), v10, z5, tool0;
	MoveL Offs(p0,31.0,50.0, 0), v10, z5, tool0;
	MoveL Offs(p0,30.0,44.0, 0), v10, z5, tool0;
	MoveL Offs(p0,30.0,43.0, 0), v10, z5, tool0;
	MoveL Offs(p0,30.0,41.0, 0), v10, z5, tool0;
	MoveL Offs(p0,29.0,40.0, 0), v10, z5, tool0;
	MoveL Offs(p0,29.0,39.0, 0), v10, z5, tool0;
	MoveL Offs(p0,28.0,38.0, 0), v10, z5, tool0;
	MoveL Offs(p0,28.0,37.0, 0), v10, z5, tool0;
	MoveL Offs(p0,27.0,37.0, 0), v10, z5, tool0;
	MoveL Offs(p0,27.0,36.0, 0), v10, z5, tool0;
	MoveL Offs(p0,26.0,35.0, 0), v10, z5, tool0;
	MoveL Offs(p0,24.0,37.0, 0), v10, z5, tool0;
	MoveL Offs(p0,23.0,39.0, 0), v10, z5, tool0;
	MoveL Offs(p0,23.0,40.0, 0), v10, z5, tool0;
	MoveL Offs(p0,22.0,40.0, 0), v10, z5, tool0;
	MoveL Offs(p0,22.0,41.0, 0), v10, z5, tool0;
	MoveL Offs(p0,22.0,41.0, 0), v10, z5, tool0;
	MoveL Offs(p0,21.0,41.0, 0), v10, z5, tool0;
	MoveL Offs(p0,20.0,44.0, 0), v10, z5, tool0;
	MoveL Offs(p0,20.0,47.0, 0), v10, z5, tool0;
	MoveL Offs(p0,21.0,49.0, 0), v10, z5, tool0;
	MoveL Offs(p0,21.0,50.0, 0), v10, z5, tool0;
	MoveL Offs(p0,21.0,50.0, 0), v10, z5, tool0;
	MoveL Offs(p0,21.0,51.0, 0), v10, z5, tool0;
	MoveL Offs(p0,21.0,52.0, 0), v10, z5, tool0;
	MoveL Offs(p0,21.0,52.0, 0), v10, z5, tool0;
	MoveL Offs(p0,21.0,53.0, 0), v10, z5, tool0;
	MoveL Offs(p0,22.0,55.0, 0), v10, z5, tool0;
	MoveL Offs(p0,22.0,55.0, 0), v10, z5, tool0;
	MoveL Offs(p0,22.0,55.0, 0), v10, z5, tool0;
	MoveL Offs(p0,22.0,55.0, 0), v10, z5, tool0;
	MoveL Offs(p0,22.0,56.0, 0), v10, z5, tool0;
	MoveL Offs(p0,22.0,56.0, 0), v10, z5, tool0;
	MoveL Offs(p0,23.0,53.0, 0), v10, z5, tool0;
	MoveL Offs(p0,23.0,53.0, 0), v10, z5, tool0;
	MoveL Offs(p0,23.0,52.0, 0), v10, z5, tool0;
	MoveL Offs(p0,24.0,54.0, 0), v10, z5, tool0;
	MoveL Offs(p0,24.0,55.0, 0), v10, z5, tool0;
	MoveL Offs(p0,24.0,56.0, 0), v10, z5, tool0;
	MoveL Offs(p0,24.0,58.0, 0), v10, z5, tool0;
	MoveL Offs(p0,24.0,59.0, 0), v10, z5, tool0;
	MoveL Offs(p0,24.0,60.0, 0), v10, z5, tool0;
	MoveL Offs(p0,24.0,61.0, 0), v10, z5, tool0;
	MoveL Offs(p0,24.0,62.0, 0), v10, z5, tool0;
	MoveL Offs(p0,26.0,62.0, 0), v10, z5, tool0;
	MoveL Offs(p0,26.0,61.0, 0), v10, z5, tool0;
	MoveL Offs(p0,26.0,60.0, 0), v10, z5, tool0;
	MoveL Offs(p0,27.0,60.0, 0), v10, z5, tool0;
	MoveL Offs(p0,27.0,59.0, 0), v10, z5, tool0;
	MoveL Offs(p0,27.0,59.0, 0), v10, z5, tool0;
	MoveL Offs(p0,28.0,61.0, 0), v10, z5, tool0;
	MoveL Offs(p0,28.0,61.0, 0), v10, z5, tool0;
	MoveL Offs(p0,29.0,62.0, 0), v10, z5, tool0;
	MoveL Offs(p0,30.0,64.0, 0), v10, z5, tool0;
	MoveL Offs(p0,30.0,64.0, 0), v10, z5, tool0;
	MoveL Offs(p0,31.0,65.0, 0), v10, z5, tool0;
	MoveL Offs(p0,31.0,65.0, 0), v10, z5, tool0;
	MoveL Offs(p0,31.0,65.0, 0), v10, z5, tool0;
	MoveL Offs(p0,31.0,64.0, 0), v10, z5, tool0;
	MoveL Offs(p0,31.0,64.0, 0), v10, z5, tool0;
	MoveL Offs(p0,31.0,63.0, 0), v10, z5, tool0;
	MoveL Offs(p0,31.0,63.0, 0), v10, z5, tool0;
	MoveJ Offs(p0,31.0,63.0, 20), v10, z1, tool0;
	MoveJ Offs(p0,19.0,57.0, 20), v10, z1, tool0;
	MoveJ Offs(p0,19.0,57.0, 0), v10, z1, tool0;
	MoveL Offs(p0,19.0,54.0, 0), v10, z5, tool0;
	MoveL Offs(p0,19.0,54.0, 0), v10, z5, tool0;
	MoveL Offs(p0,19.0,54.0, 0), v10, z5, tool0;
	MoveL Offs(p0,19.0,54.0, 0), v10, z5, tool0;
	MoveL Offs(p0,19.0,54.0, 0), v10, z5, tool0;
	MoveL Offs(p0,17.0,54.0, 0), v10, z5, tool0;
	MoveL Offs(p0,17.0,58.0, 0), v10, z5, tool0;
	MoveL Offs(p0,18.0,58.0, 0), v10, z5, tool0;
	MoveL Offs(p0,18.0,59.0, 0), v10, z5, tool0;
	MoveL Offs(p0,18.0,59.0, 0), v10, z5, tool0;
	MoveL Offs(p0,18.0,59.0, 0), v10, z5, tool0;
	MoveL Offs(p0,19.0,58.0, 0), v10, z5, tool0;
	MoveL Offs(p0,19.0,57.0, 0), v10, z5, tool0;
	MoveL Offs(p0,19.0,57.0, 0), v10, z5, tool0;
	MoveL Offs(p0,19.0,57.0, 0), v10, z5, tool0;
	MoveJ Offs(p0,19.0,57.0, 20), v10, z1, tool0;
	MoveJ Offs(p0,5.0,59.0, 20), v10, z1, tool0;
	MoveJ Offs(p0,5.0,59.0, 0), v10, z1, tool0;
	MoveL Offs(p0,5.0,56.0, 0), v10, z5, tool0;
	MoveL Offs(p0,5.0,56.0, 0), v10, z5, tool0;
	MoveL Offs(p0,6.0,55.0, 0), v10, z5, tool0;
	MoveL Offs(p0,6.0,55.0, 0), v10, z5, tool0;
	MoveL Offs(p0,6.0,53.0, 0), v10, z5, tool0;
	MoveL Offs(p0,6.0,52.0, 0), v10, z5, tool0;
	MoveL Offs(p0,6.0,52.0, 0), v10, z5, tool0;
	MoveL Offs(p0,6.0,52.0, 0), v10, z5, tool0;
	MoveL Offs(p0,6.0,51.0, 0), v10, z5, tool0;
	MoveL Offs(p0,5.0,51.0, 0), v10, z5, tool0;
	MoveL Offs(p0,5.0,51.0, 0), v10, z5, tool0;
	MoveL Offs(p0,3.0,49.0, 0), v10, z5, tool0;
	MoveL Offs(p0,3.0,48.0, 0), v10, z5, tool0;
	MoveL Offs(p0,3.0,49.0, 0), v10, z5, tool0;
	MoveL Offs(p0,2.0,51.0, 0), v10, z5, tool0;
	MoveL Offs(p0,2.0,53.0, 0), v10, z5, tool0;
	MoveL Offs(p0,2.0,54.0, 0), v10, z5, tool0;
	MoveL Offs(p0,3.0,55.0, 0), v10, z5, tool0;
	MoveL Offs(p0,3.0,56.0, 0), v10, z5, tool0;
	MoveL Offs(p0,3.0,57.0, 0), v10, z5, tool0;
	MoveL Offs(p0,3.0,58.0, 0), v10, z5, tool0;
	MoveL Offs(p0,3.0,58.0, 0), v10, z5, tool0;
	MoveL Offs(p0,5.0,59.0, 0), v10, z5, tool0;
	MoveJ Offs(p0,5.0,59.0, 20), v10, z1, tool0;
	MoveJ Offs(p0,69.0,53.0, 20), v10, z1, tool0;
	MoveJ Offs(p0,69.0,53.0, 0), v10, z1, tool0;
	MoveL Offs(p0,69.0,51.0, 0), v10, z5, tool0;
	MoveL Offs(p0,69.0,50.0, 0), v10, z5, tool0;
	MoveL Offs(p0,69.0,50.0, 0), v10, z5, tool0;
	MoveL Offs(p0,69.0,49.0, 0), v10, z5, tool0;
	MoveL Offs(p0,69.0,49.0, 0), v10, z5, tool0;
	MoveL Offs(p0,69.0,48.0, 0), v10, z5, tool0;
	MoveL Offs(p0,70.0,48.0, 0), v10, z5, tool0;
	MoveL Offs(p0,70.0,47.0, 0), v10, z5, tool0;
	MoveL Offs(p0,71.0,45.0, 0), v10, z5, tool0;
	MoveL Offs(p0,71.0,44.0, 0), v10, z5, tool0;
	MoveL Offs(p0,71.0,44.0, 0), v10, z5, tool0;
	MoveL Offs(p0,72.0,44.0, 0), v10, z5, tool0;
	MoveL Offs(p0,72.0,43.0, 0), v10, z5, tool0;
	MoveL Offs(p0,72.0,43.0, 0), v10, z5, tool0;
	MoveL Offs(p0,73.0,43.0, 0), v10, z5, tool0;
	MoveL Offs(p0,73.0,43.0, 0), v10, z5, tool0;
	MoveL Offs(p0,74.0,45.0, 0), v10, z5, tool0;
	MoveL Offs(p0,74.0,46.0, 0), v10, z5, tool0;
	MoveL Offs(p0,74.0,47.0, 0), v10, z5, tool0;
	MoveL Offs(p0,75.0,50.0, 0), v10, z5, tool0;
	MoveL Offs(p0,75.0,50.0, 0), v10, z5, tool0;
	MoveL Offs(p0,75.0,51.0, 0), v10, z5, tool0;
	MoveL Offs(p0,75.0,51.0, 0), v10, z5, tool0;
	MoveL Offs(p0,75.0,52.0, 0), v10, z5, tool0;
	MoveL Offs(p0,75.0,52.0, 0), v10, z5, tool0;
	MoveL Offs(p0,75.0,52.0, 0), v10, z5, tool0;
	MoveL Offs(p0,75.0,53.0, 0), v10, z5, tool0;
	MoveL Offs(p0,78.0,52.0, 0), v10, z5, tool0;
	MoveL Offs(p0,80.0,51.0, 0), v10, z5, tool0;
	MoveL Offs(p0,80.0,50.0, 0), v10, z5, tool0;
	MoveL Offs(p0,79.0,48.0, 0), v10, z5, tool0;
	MoveL Offs(p0,78.0,46.0, 0), v10, z5, tool0;
	MoveL Offs(p0,78.0,45.0, 0), v10, z5, tool0;
	MoveL Offs(p0,78.0,43.0, 0), v10, z5, tool0;
	MoveL Offs(p0,78.0,41.0, 0), v10, z5, tool0;
	MoveL Offs(p0,78.0,40.0, 0), v10, z5, tool0;
	MoveL Offs(p0,78.0,38.0, 0), v10, z5, tool0;
	MoveL Offs(p0,79.0,37.0, 0), v10, z5, tool0;
	MoveL Offs(p0,79.0,35.0, 0), v10, z5, tool0;
	MoveL Offs(p0,74.0,38.0, 0), v10, z5, tool0;
	MoveL Offs(p0,73.0,40.0, 0), v10, z5, tool0;
	MoveL Offs(p0,72.0,41.0, 0), v10, z5, tool0;
	MoveL Offs(p0,70.0,43.0, 0), v10, z5, tool0;
	MoveL Offs(p0,69.0,45.0, 0), v10, z5, tool0;
	MoveL Offs(p0,69.0,47.0, 0), v10, z5, tool0;
	MoveL Offs(p0,68.0,49.0, 0), v10, z5, tool0;
	MoveL Offs(p0,68.0,51.0, 0), v10, z5, tool0;
	MoveL Offs(p0,68.0,53.0, 0), v10, z5, tool0;
	MoveL Offs(p0,68.0,56.0, 0), v10, z5, tool0;
	MoveL Offs(p0,68.0,56.0, 0), v10, z5, tool0;
	MoveL Offs(p0,68.0,57.0, 0), v10, z5, tool0;
	MoveL Offs(p0,68.0,57.0, 0), v10, z5, tool0;
	MoveL Offs(p0,68.0,58.0, 0), v10, z5, tool0;
	MoveL Offs(p0,69.0,58.0, 0), v10, z5, tool0;
	MoveL Offs(p0,69.0,58.0, 0), v10, z5, tool0;
	MoveL Offs(p0,69.0,58.0, 0), v10, z5, tool0;
	MoveL Offs(p0,69.0,56.0, 0), v10, z5, tool0;
	MoveL Offs(p0,69.0,55.0, 0), v10, z5, tool0;
	MoveL Offs(p0,69.0,54.0, 0), v10, z5, tool0;
	MoveL Offs(p0,69.0,53.0, 0), v10, z5, tool0;
	MoveL Offs(p0,69.0,53.0, 0), v10, z5, tool0;
	MoveJ Offs(p0,69.0,53.0, 20), v10, z1, tool0;
	MoveJ Offs(p0,105.0,57.0, 20), v10, z1, tool0;
	MoveJ Offs(p0,105.0,57.0, 0), v10, z1, tool0;
	MoveL Offs(p0,106.0,55.0, 0), v10, z5, tool0;
	MoveL Offs(p0,107.0,54.0, 0), v10, z5, tool0;
	MoveL Offs(p0,107.0,52.0, 0), v10, z5, tool0;
	MoveL Offs(p0,107.0,51.0, 0), v10, z5, tool0;
	MoveL Offs(p0,107.0,49.0, 0), v10, z5, tool0;
	MoveL Offs(p0,107.0,48.0, 0), v10, z5, tool0;
	MoveL Offs(p0,107.0,46.0, 0), v10, z5, tool0;
	MoveL Offs(p0,107.0,45.0, 0), v10, z5, tool0;
	MoveL Offs(p0,106.0,42.0, 0), v10, z5, tool0;
	MoveL Offs(p0,105.0,41.0, 0), v10, z5, tool0;
	MoveL Offs(p0,105.0,40.0, 0), v10, z5, tool0;
	MoveL Offs(p0,104.0,39.0, 0), v10, z5, tool0;
	MoveL Offs(p0,103.0,38.0, 0), v10, z5, tool0;
	MoveL Offs(p0,102.0,37.0, 0), v10, z5, tool0;
	MoveL Offs(p0,101.0,36.0, 0), v10, z5, tool0;
	MoveL Offs(p0,100.0,35.0, 0), v10, z5, tool0;
	MoveL Offs(p0,99.0,35.0, 0), v10, z5, tool0;
	MoveL Offs(p0,96.0,34.0, 0), v10, z5, tool0;
	MoveL Offs(p0,96.0,33.0, 0), v10, z5, tool0;
	MoveL Offs(p0,95.0,33.0, 0), v10, z5, tool0;
	MoveL Offs(p0,94.0,33.0, 0), v10, z5, tool0;
	MoveL Offs(p0,92.0,33.0, 0), v10, z5, tool0;
	MoveL Offs(p0,91.0,33.0, 0), v10, z5, tool0;
	MoveL Offs(p0,91.0,32.0, 0), v10, z5, tool0;
	MoveL Offs(p0,90.0,32.0, 0), v10, z5, tool0;
	MoveL Offs(p0,87.0,33.0, 0), v10, z5, tool0;
	MoveL Offs(p0,86.0,33.0, 0), v10, z5, tool0;
	MoveL Offs(p0,84.0,33.0, 0), v10, z5, tool0;
	MoveL Offs(p0,84.0,33.0, 0), v10, z5, tool0;
	MoveL Offs(p0,83.0,33.0, 0), v10, z5, tool0;
	MoveL Offs(p0,82.0,34.0, 0), v10, z5, tool0;
	MoveL Offs(p0,81.0,34.0, 0), v10, z5, tool0;
	MoveL Offs(p0,81.0,34.0, 0), v10, z5, tool0;
	MoveL Offs(p0,80.0,37.0, 0), v10, z5, tool0;
	MoveL Offs(p0,79.0,39.0, 0), v10, z5, tool0;
	MoveL Offs(p0,79.0,40.0, 0), v10, z5, tool0;
	MoveL Offs(p0,79.0,42.0, 0), v10, z5, tool0;
	MoveL Offs(p0,79.0,44.0, 0), v10, z5, tool0;
	MoveL Offs(p0,79.0,45.0, 0), v10, z5, tool0;
	MoveL Offs(p0,79.0,47.0, 0), v10, z5, tool0;
	MoveL Offs(p0,80.0,48.0, 0), v10, z5, tool0;
	MoveL Offs(p0,81.0,50.0, 0), v10, z5, tool0;
	MoveL Offs(p0,81.0,51.0, 0), v10, z5, tool0;
	MoveL Offs(p0,82.0,51.0, 0), v10, z5, tool0;
	MoveL Offs(p0,83.0,51.0, 0), v10, z5, tool0;
	MoveL Offs(p0,84.0,51.0, 0), v10, z5, tool0;
	MoveL Offs(p0,85.0,51.0, 0), v10, z5, tool0;
	MoveL Offs(p0,86.0,51.0, 0), v10, z5, tool0;
	MoveL Offs(p0,88.0,51.0, 0), v10, z5, tool0;
	MoveL Offs(p0,89.0,51.0, 0), v10, z5, tool0;
	MoveL Offs(p0,90.0,51.0, 0), v10, z5, tool0;
	MoveL Offs(p0,90.0,51.0, 0), v10, z5, tool0;
	MoveL Offs(p0,91.0,51.0, 0), v10, z5, tool0;
	MoveL Offs(p0,92.0,51.0, 0), v10, z5, tool0;
	MoveL Offs(p0,92.0,51.0, 0), v10, z5, tool0;
	MoveL Offs(p0,93.0,51.0, 0), v10, z5, tool0;
	MoveL Offs(p0,95.0,52.0, 0), v10, z5, tool0;
	MoveL Offs(p0,96.0,52.0, 0), v10, z5, tool0;
	MoveL Offs(p0,97.0,53.0, 0), v10, z5, tool0;
	MoveL Offs(p0,98.0,53.0, 0), v10, z5, tool0;
	MoveL Offs(p0,99.0,54.0, 0), v10, z5, tool0;
	MoveL Offs(p0,100.0,54.0, 0), v10, z5, tool0;
	MoveL Offs(p0,100.0,55.0, 0), v10, z5, tool0;
	MoveL Offs(p0,101.0,55.0, 0), v10, z5, tool0;
	MoveL Offs(p0,102.0,56.0, 0), v10, z5, tool0;
	MoveL Offs(p0,104.0,58.0, 0), v10, z5, tool0;
	MoveL Offs(p0,104.0,58.0, 0), v10, z5, tool0;
	MoveL Offs(p0,105.0,57.0, 0), v10, z5, tool0;
	MoveJ Offs(p0,105.0,57.0, 20), v10, z1, tool0;
	MoveJ Offs(p0,74.0,51.0, 20), v10, z1, tool0;
	MoveJ Offs(p0,74.0,51.0, 0), v10, z1, tool0;
	MoveL Offs(p0,74.0,49.0, 0), v10, z5, tool0;
	MoveL Offs(p0,74.0,48.0, 0), v10, z5, tool0;
	MoveL Offs(p0,74.0,48.0, 0), v10, z5, tool0;
	MoveL Offs(p0,74.0,47.0, 0), v10, z5, tool0;
	MoveL Offs(p0,74.0,47.0, 0), v10, z5, tool0;
	MoveL Offs(p0,74.0,46.0, 0), v10, z5, tool0;
	MoveL Offs(p0,73.0,44.0, 0), v10, z5, tool0;
	MoveL Offs(p0,73.0,44.0, 0), v10, z5, tool0;
	MoveL Offs(p0,73.0,44.0, 0), v10, z5, tool0;
	MoveL Offs(p0,73.0,43.0, 0), v10, z5, tool0;
	MoveL Offs(p0,73.0,43.0, 0), v10, z5, tool0;
	MoveL Offs(p0,72.0,43.0, 0), v10, z5, tool0;
	MoveL Offs(p0,72.0,44.0, 0), v10, z5, tool0;
	MoveL Offs(p0,71.0,46.0, 0), v10, z5, tool0;
	MoveL Offs(p0,70.0,47.0, 0), v10, z5, tool0;
	MoveL Offs(p0,70.0,48.0, 0), v10, z5, tool0;
	MoveL Offs(p0,70.0,50.0, 0), v10, z5, tool0;
	MoveL Offs(p0,70.0,51.0, 0), v10, z5, tool0;
	MoveL Offs(p0,70.0,53.0, 0), v10, z5, tool0;
	MoveL Offs(p0,70.0,54.0, 0), v10, z5, tool0;
	MoveL Offs(p0,70.0,55.0, 0), v10, z5, tool0;
	MoveL Offs(p0,70.0,56.0, 0), v10, z5, tool0;
	MoveL Offs(p0,73.0,55.0, 0), v10, z5, tool0;
	MoveL Offs(p0,75.0,54.0, 0), v10, z5, tool0;
	MoveL Offs(p0,74.0,51.0, 0), v10, z5, tool0;
	MoveL Offs(p0,74.0,51.0, 0), v10, z5, tool0;
	MoveJ Offs(p0,74.0,51.0, 20), v10, z1, tool0;
	MoveJ Offs(p0,19.0,52.0, 20), v10, z1, tool0;
	MoveJ Offs(p0,19.0,52.0, 0), v10, z1, tool0;
	MoveL Offs(p0,20.0,50.0, 0), v10, z5, tool0;
	MoveL Offs(p0,20.0,49.0, 0), v10, z5, tool0;
	MoveL Offs(p0,20.0,48.0, 0), v10, z5, tool0;
	MoveL Offs(p0,20.0,48.0, 0), v10, z5, tool0;
	MoveL Offs(p0,19.0,45.0, 0), v10, z5, tool0;
	MoveL Offs(p0,19.0,45.0, 0), v10, z5, tool0;
	MoveL Offs(p0,18.0,45.0, 0), v10, z5, tool0;
	MoveL Offs(p0,18.0,44.0, 0), v10, z5, tool0;
	MoveL Offs(p0,18.0,44.0, 0), v10, z5, tool0;
	MoveL Offs(p0,17.0,44.0, 0), v10, z5, tool0;
	MoveL Offs(p0,17.0,43.0, 0), v10, z5, tool0;
	MoveL Offs(p0,16.0,43.0, 0), v10, z5, tool0;
	MoveL Offs(p0,14.0,42.0, 0), v10, z5, tool0;
	MoveL Offs(p0,14.0,42.0, 0), v10, z5, tool0;
	MoveL Offs(p0,13.0,41.0, 0), v10, z5, tool0;
	MoveL Offs(p0,13.0,41.0, 0), v10, z5, tool0;
	MoveL Offs(p0,13.0,41.0, 0), v10, z5, tool0;
	MoveL Offs(p0,12.0,40.0, 0), v10, z5, tool0;
	MoveL Offs(p0,10.0,39.0, 0), v10, z5, tool0;
	MoveL Offs(p0,9.0,41.0, 0), v10, z5, tool0;
	MoveL Offs(p0,8.0,43.0, 0), v10, z5, tool0;
	MoveL Offs(p0,8.0,43.0, 0), v10, z5, tool0;
	MoveL Offs(p0,7.0,44.0, 0), v10, z5, tool0;
	MoveL Offs(p0,7.0,44.0, 0), v10, z5, tool0;
	MoveL Offs(p0,6.0,44.0, 0), v10, z5, tool0;
	MoveL Offs(p0,6.0,45.0, 0), v10, z5, tool0;
	MoveL Offs(p0,6.0,45.0, 0), v10, z5, tool0;
	MoveL Offs(p0,5.0,45.0, 0), v10, z5, tool0;
	MoveL Offs(p0,5.0,41.0, 0), v10, z5, tool0;
	MoveL Offs(p0,5.0,40.0, 0), v10, z5, tool0;
	MoveL Offs(p0,5.0,39.0, 0), v10, z5, tool0;
	MoveL Offs(p0,5.0,38.0, 0), v10, z5, tool0;
	MoveL Offs(p0,6.0,37.0, 0), v10, z5, tool0;
	MoveL Offs(p0,6.0,36.0, 0), v10, z5, tool0;
	MoveL Offs(p0,6.0,35.0, 0), v10, z5, tool0;
	MoveL Offs(p0,7.0,34.0, 0), v10, z5, tool0;
	MoveL Offs(p0,8.0,32.0, 0), v10, z5, tool0;
	MoveL Offs(p0,8.0,32.0, 0), v10, z5, tool0;
	MoveL Offs(p0,8.0,32.0, 0), v10, z5, tool0;
	MoveL Offs(p0,8.0,31.0, 0), v10, z5, tool0;
	MoveL Offs(p0,8.0,31.0, 0), v10, z5, tool0;
	MoveL Offs(p0,5.0,35.0, 0), v10, z5, tool0;
	MoveL Offs(p0,5.0,35.0, 0), v10, z5, tool0;
	MoveL Offs(p0,4.0,36.0, 0), v10, z5, tool0;
	MoveL Offs(p0,4.0,37.0, 0), v10, z5, tool0;
	MoveL Offs(p0,4.0,38.0, 0), v10, z5, tool0;
	MoveL Offs(p0,4.0,39.0, 0), v10, z5, tool0;
	MoveL Offs(p0,3.0,40.0, 0), v10, z5, tool0;
	MoveL Offs(p0,3.0,41.0, 0), v10, z5, tool0;
	MoveL Offs(p0,3.0,43.0, 0), v10, z5, tool0;
	MoveL Offs(p0,3.0,45.0, 0), v10, z5, tool0;
	MoveL Offs(p0,4.0,46.0, 0), v10, z5, tool0;
	MoveL Offs(p0,4.0,47.0, 0), v10, z5, tool0;
	MoveL Offs(p0,5.0,48.0, 0), v10, z5, tool0;
	MoveL Offs(p0,5.0,49.0, 0), v10, z5, tool0;
	MoveL Offs(p0,6.0,50.0, 0), v10, z5, tool0;
	MoveL Offs(p0,7.0,51.0, 0), v10, z5, tool0;
	MoveL Offs(p0,9.0,52.0, 0), v10, z5, tool0;
	MoveL Offs(p0,11.0,53.0, 0), v10, z5, tool0;
	MoveL Offs(p0,12.0,53.0, 0), v10, z5, tool0;
	MoveL Offs(p0,13.0,53.0, 0), v10, z5, tool0;
	MoveL Offs(p0,14.0,53.0, 0), v10, z5, tool0;
	MoveL Offs(p0,15.0,53.0, 0), v10, z5, tool0;
	MoveL Offs(p0,16.0,53.0, 0), v10, z5, tool0;
	MoveL Offs(p0,17.0,53.0, 0), v10, z5, tool0;
	MoveL Offs(p0,18.0,52.0, 0), v10, z5, tool0;
	MoveL Offs(p0,19.0,52.0, 0), v10, z5, tool0;
	MoveL Offs(p0,19.0,52.0, 0), v10, z5, tool0;
	MoveJ Offs(p0,19.0,52.0, 20), v10, z1, tool0;
	MoveJ Offs(p0,68.0,44.0, 20), v10, z1, tool0;
	MoveJ Offs(p0,68.0,44.0, 0), v10, z1, tool0;
	MoveL Offs(p0,68.0,42.0, 0), v10, z5, tool0;
	MoveL Offs(p0,67.0,42.0, 0), v10, z5, tool0;
	MoveL Offs(p0,66.0,39.0, 0), v10, z5, tool0;
	MoveL Offs(p0,65.0,37.0, 0), v10, z5, tool0;
	MoveL Offs(p0,65.0,36.0, 0), v10, z5, tool0;
	MoveL Offs(p0,64.0,34.0, 0), v10, z5, tool0;
	MoveL Offs(p0,64.0,33.0, 0), v10, z5, tool0;
	MoveL Offs(p0,65.0,31.0, 0), v10, z5, tool0;
	MoveL Offs(p0,65.0,30.0, 0), v10, z5, tool0;
	MoveL Offs(p0,66.0,30.0, 0), v10, z5, tool0;
	MoveL Offs(p0,66.0,30.0, 0), v10, z5, tool0;
	MoveL Offs(p0,69.0,31.0, 0), v10, z5, tool0;
	MoveL Offs(p0,69.0,32.0, 0), v10, z5, tool0;
	MoveL Offs(p0,70.0,32.0, 0), v10, z5, tool0;
	MoveL Offs(p0,70.0,33.0, 0), v10, z5, tool0;
	MoveL Offs(p0,72.0,35.0, 0), v10, z5, tool0;
	MoveL Offs(p0,73.0,35.0, 0), v10, z5, tool0;
	MoveL Offs(p0,73.0,36.0, 0), v10, z5, tool0;
	MoveL Offs(p0,74.0,36.0, 0), v10, z5, tool0;
	MoveL Offs(p0,74.0,36.0, 0), v10, z5, tool0;
	MoveL Offs(p0,75.0,36.0, 0), v10, z5, tool0;
	MoveL Offs(p0,76.0,36.0, 0), v10, z5, tool0;
	MoveL Offs(p0,76.0,35.0, 0), v10, z5, tool0;
	MoveL Offs(p0,77.0,35.0, 0), v10, z5, tool0;
	MoveL Offs(p0,80.0,33.0, 0), v10, z5, tool0;
	MoveL Offs(p0,78.0,33.0, 0), v10, z5, tool0;
	MoveL Offs(p0,74.0,30.0, 0), v10, z5, tool0;
	MoveL Offs(p0,72.0,27.0, 0), v10, z5, tool0;
	MoveL Offs(p0,72.0,26.0, 0), v10, z5, tool0;
	MoveL Offs(p0,72.0,25.0, 0), v10, z5, tool0;
	MoveL Offs(p0,71.0,24.0, 0), v10, z5, tool0;
	MoveL Offs(p0,71.0,24.0, 0), v10, z5, tool0;
	MoveL Offs(p0,71.0,23.0, 0), v10, z5, tool0;
	MoveL Offs(p0,71.0,22.0, 0), v10, z5, tool0;
	MoveL Offs(p0,71.0,21.0, 0), v10, z5, tool0;
	MoveL Offs(p0,68.0,21.0, 0), v10, z5, tool0;
	MoveL Offs(p0,68.0,22.0, 0), v10, z5, tool0;
	MoveL Offs(p0,67.0,22.0, 0), v10, z5, tool0;
	MoveL Offs(p0,66.0,23.0, 0), v10, z5, tool0;
	MoveL Offs(p0,66.0,24.0, 0), v10, z5, tool0;
	MoveL Offs(p0,65.0,25.0, 0), v10, z5, tool0;
	MoveL Offs(p0,64.0,27.0, 0), v10, z5, tool0;
	MoveL Offs(p0,64.0,28.0, 0), v10, z5, tool0;
	MoveL Offs(p0,63.0,29.0, 0), v10, z5, tool0;
	MoveL Offs(p0,63.0,30.0, 0), v10, z5, tool0;
	MoveL Offs(p0,63.0,31.0, 0), v10, z5, tool0;
	MoveL Offs(p0,63.0,32.0, 0), v10, z5, tool0;
	MoveL Offs(p0,63.0,34.0, 0), v10, z5, tool0;
	MoveL Offs(p0,63.0,35.0, 0), v10, z5, tool0;
	MoveL Offs(p0,63.0,37.0, 0), v10, z5, tool0;
	MoveL Offs(p0,63.0,38.0, 0), v10, z5, tool0;
	MoveL Offs(p0,63.0,39.0, 0), v10, z5, tool0;
	MoveL Offs(p0,64.0,40.0, 0), v10, z5, tool0;
	MoveL Offs(p0,64.0,41.0, 0), v10, z5, tool0;
	MoveL Offs(p0,64.0,41.0, 0), v10, z5, tool0;
	MoveL Offs(p0,65.0,42.0, 0), v10, z5, tool0;
	MoveL Offs(p0,65.0,43.0, 0), v10, z5, tool0;
	MoveL Offs(p0,66.0,44.0, 0), v10, z5, tool0;
	MoveL Offs(p0,68.0,45.0, 0), v10, z5, tool0;
	MoveL Offs(p0,68.0,44.0, 0), v10, z5, tool0;
	MoveL Offs(p0,68.0,44.0, 0), v10, z5, tool0;
	MoveJ Offs(p0,68.0,44.0, 20), v10, z1, tool0;
	MoveJ Offs(p0,7.0,43.0, 20), v10, z1, tool0;
	MoveJ Offs(p0,7.0,43.0, 0), v10, z1, tool0;
	MoveL Offs(p0,9.0,41.0, 0), v10, z5, tool0;
	MoveL Offs(p0,9.0,40.0, 0), v10, z5, tool0;
	MoveL Offs(p0,9.0,40.0, 0), v10, z5, tool0;
	MoveL Offs(p0,9.0,40.0, 0), v10, z5, tool0;
	MoveL Offs(p0,10.0,38.0, 0), v10, z5, tool0;
	MoveL Offs(p0,9.0,36.0, 0), v10, z5, tool0;
	MoveL Offs(p0,8.0,33.0, 0), v10, z5, tool0;
	MoveL Offs(p0,8.0,33.0, 0), v10, z5, tool0;
	MoveL Offs(p0,8.0,33.0, 0), v10, z5, tool0;
	MoveL Offs(p0,8.0,33.0, 0), v10, z5, tool0;
	MoveL Offs(p0,7.0,36.0, 0), v10, z5, tool0;
	MoveL Offs(p0,6.0,37.0, 0), v10, z5, tool0;
	MoveL Offs(p0,6.0,37.0, 0), v10, z5, tool0;
	MoveL Offs(p0,6.0,38.0, 0), v10, z5, tool0;
	MoveL Offs(p0,6.0,39.0, 0), v10, z5, tool0;
	MoveL Offs(p0,5.0,41.0, 0), v10, z5, tool0;
	MoveL Offs(p0,5.0,42.0, 0), v10, z5, tool0;
	MoveL Offs(p0,5.0,43.0, 0), v10, z5, tool0;
	MoveL Offs(p0,5.0,43.0, 0), v10, z5, tool0;
	MoveL Offs(p0,5.0,44.0, 0), v10, z5, tool0;
	MoveL Offs(p0,5.0,44.0, 0), v10, z5, tool0;
	MoveL Offs(p0,5.0,44.0, 0), v10, z5, tool0;
	MoveL Offs(p0,5.0,44.0, 0), v10, z5, tool0;
	MoveL Offs(p0,7.0,43.0, 0), v10, z5, tool0;
	MoveJ Offs(p0,7.0,43.0, 20), v10, z1, tool0;
	MoveJ Offs(p0,21.0,40.0, 20), v10, z1, tool0;
	MoveJ Offs(p0,21.0,40.0, 0), v10, z1, tool0;
	MoveL Offs(p0,22.0,38.0, 0), v10, z5, tool0;
	MoveL Offs(p0,23.0,37.0, 0), v10, z5, tool0;
	MoveL Offs(p0,23.0,37.0, 0), v10, z5, tool0;
	MoveL Offs(p0,24.0,36.0, 0), v10, z5, tool0;
	MoveL Offs(p0,24.0,35.0, 0), v10, z5, tool0;
	MoveL Offs(p0,25.0,35.0, 0), v10, z5, tool0;
	MoveL Offs(p0,25.0,34.0, 0), v10, z5, tool0;
	MoveL Offs(p0,25.0,34.0, 0), v10, z5, tool0;
	MoveL Offs(p0,17.0,32.0, 0), v10, z5, tool0;
	MoveL Offs(p0,16.0,33.0, 0), v10, z5, tool0;
	MoveL Offs(p0,16.0,33.0, 0), v10, z5, tool0;
	MoveL Offs(p0,15.0,34.0, 0), v10, z5, tool0;
	MoveL Offs(p0,14.0,34.0, 0), v10, z5, tool0;
	MoveL Offs(p0,14.0,34.0, 0), v10, z5, tool0;
	MoveL Offs(p0,13.0,34.0, 0), v10, z5, tool0;
	MoveL Offs(p0,12.0,32.0, 0), v10, z5, tool0;
	MoveL Offs(p0,12.0,31.0, 0), v10, z5, tool0;
	MoveL Offs(p0,12.0,30.0, 0), v10, z5, tool0;
	MoveL Offs(p0,13.0,29.0, 0), v10, z5, tool0;
	MoveL Offs(p0,14.0,27.0, 0), v10, z5, tool0;
	MoveL Offs(p0,15.0,26.0, 0), v10, z5, tool0;
	MoveL Offs(p0,16.0,24.0, 0), v10, z5, tool0;
	MoveL Offs(p0,18.0,22.0, 0), v10, z5, tool0;
	MoveL Offs(p0,18.0,22.0, 0), v10, z5, tool0;
	MoveL Offs(p0,18.0,22.0, 0), v10, z5, tool0;
	MoveL Offs(p0,18.0,21.0, 0), v10, z5, tool0;
	MoveL Offs(p0,18.0,21.0, 0), v10, z5, tool0;
	MoveL Offs(p0,18.0,21.0, 0), v10, z5, tool0;
	MoveL Offs(p0,18.0,18.0, 0), v10, z5, tool0;
	MoveL Offs(p0,19.0,18.0, 0), v10, z5, tool0;
	MoveL Offs(p0,19.0,18.0, 0), v10, z5, tool0;
	MoveL Offs(p0,19.0,17.0, 0), v10, z5, tool0;
	MoveL Offs(p0,16.0,18.0, 0), v10, z5, tool0;
	MoveL Offs(p0,16.0,18.0, 0), v10, z5, tool0;
	MoveL Offs(p0,15.0,19.0, 0), v10, z5, tool0;
	MoveL Offs(p0,15.0,19.0, 0), v10, z5, tool0;
	MoveL Offs(p0,13.0,21.0, 0), v10, z5, tool0;
	MoveL Offs(p0,12.0,22.0, 0), v10, z5, tool0;
	MoveL Offs(p0,11.0,23.0, 0), v10, z5, tool0;
	MoveL Offs(p0,11.0,24.0, 0), v10, z5, tool0;
	MoveL Offs(p0,10.0,26.0, 0), v10, z5, tool0;
	MoveL Offs(p0,10.0,27.0, 0), v10, z5, tool0;
	MoveL Offs(p0,10.0,28.0, 0), v10, z5, tool0;
	MoveL Offs(p0,9.0,29.0, 0), v10, z5, tool0;
	MoveL Offs(p0,9.0,30.0, 0), v10, z5, tool0;
	MoveL Offs(p0,10.0,33.0, 0), v10, z5, tool0;
	MoveL Offs(p0,10.0,34.0, 0), v10, z5, tool0;
	MoveL Offs(p0,10.0,35.0, 0), v10, z5, tool0;
	MoveL Offs(p0,10.0,36.0, 0), v10, z5, tool0;
	MoveL Offs(p0,11.0,36.0, 0), v10, z5, tool0;
	MoveL Offs(p0,11.0,37.0, 0), v10, z5, tool0;
	MoveL Offs(p0,12.0,38.0, 0), v10, z5, tool0;
	MoveL Offs(p0,12.0,39.0, 0), v10, z5, tool0;
	MoveL Offs(p0,15.0,41.0, 0), v10, z5, tool0;
	MoveL Offs(p0,15.0,41.0, 0), v10, z5, tool0;
	MoveL Offs(p0,16.0,42.0, 0), v10, z5, tool0;
	MoveL Offs(p0,17.0,42.0, 0), v10, z5, tool0;
	MoveL Offs(p0,17.0,42.0, 0), v10, z5, tool0;
	MoveL Offs(p0,18.0,42.0, 0), v10, z5, tool0;
	MoveL Offs(p0,18.0,42.0, 0), v10, z5, tool0;
	MoveL Offs(p0,20.0,41.0, 0), v10, z5, tool0;
	MoveL Offs(p0,21.0,40.0, 0), v10, z5, tool0;
	MoveL Offs(p0,21.0,40.0, 0), v10, z5, tool0;
	MoveJ Offs(p0,21.0,40.0, 20), v10, z1, tool0;
	MoveJ Offs(p0,70.0,41.0, 20), v10, z1, tool0;
	MoveJ Offs(p0,70.0,41.0, 0), v10, z1, tool0;
	MoveL Offs(p0,72.0,39.0, 0), v10, z5, tool0;
	MoveL Offs(p0,72.0,39.0, 0), v10, z5, tool0;
	MoveL Offs(p0,73.0,38.0, 0), v10, z5, tool0;
	MoveL Offs(p0,74.0,37.0, 0), v10, z5, tool0;
	MoveL Offs(p0,70.0,34.0, 0), v10, z5, tool0;
	MoveL Offs(p0,68.0,32.0, 0), v10, z5, tool0;
	MoveL Offs(p0,68.0,31.0, 0), v10, z5, tool0;
	MoveL Offs(p0,67.0,31.0, 0), v10, z5, tool0;
	MoveL Offs(p0,67.0,31.0, 0), v10, z5, tool0;
	MoveL Offs(p0,67.0,31.0, 0), v10, z5, tool0;
	MoveL Offs(p0,66.0,30.0, 0), v10, z5, tool0;
	MoveL Offs(p0,66.0,30.0, 0), v10, z5, tool0;
	MoveL Offs(p0,65.0,33.0, 0), v10, z5, tool0;
	MoveL Offs(p0,65.0,35.0, 0), v10, z5, tool0;
	MoveL Offs(p0,66.0,36.0, 0), v10, z5, tool0;
	MoveL Offs(p0,66.0,37.0, 0), v10, z5, tool0;
	MoveL Offs(p0,66.0,39.0, 0), v10, z5, tool0;
	MoveL Offs(p0,67.0,40.0, 0), v10, z5, tool0;
	MoveL Offs(p0,68.0,41.0, 0), v10, z5, tool0;
	MoveL Offs(p0,70.0,41.0, 0), v10, z5, tool0;
	MoveJ Offs(p0,70.0,41.0, 20), v10, z1, tool0;
	MoveJ Offs(p0,32.0,37.0, 20), v10, z1, tool0;
	MoveJ Offs(p0,32.0,37.0, 0), v10, z1, tool0;
	MoveL Offs(p0,29.0,35.0, 0), v10, z5, tool0;
	MoveL Offs(p0,29.0,35.0, 0), v10, z5, tool0;
	MoveL Offs(p0,29.0,38.0, 0), v10, z5, tool0;
	MoveL Offs(p0,29.0,38.0, 0), v10, z5, tool0;
	MoveL Offs(p0,32.0,37.0, 0), v10, z5, tool0;
	MoveJ Offs(p0,32.0,37.0, 20), v10, z1, tool0;
	MoveJ Offs(p0,61.0,34.0, 20), v10, z1, tool0;
	MoveJ Offs(p0,61.0,34.0, 0), v10, z1, tool0;
	MoveL Offs(p0,61.0,32.0, 0), v10, z5, tool0;
	MoveL Offs(p0,61.0,32.0, 0), v10, z5, tool0;
	MoveL Offs(p0,61.0,32.0, 0), v10, z5, tool0;
	MoveL Offs(p0,58.0,31.0, 0), v10, z5, tool0;
	MoveL Offs(p0,57.0,31.0, 0), v10, z5, tool0;
	MoveL Offs(p0,57.0,30.0, 0), v10, z5, tool0;
	MoveL Offs(p0,56.0,30.0, 0), v10, z5, tool0;
	MoveL Offs(p0,55.0,29.0, 0), v10, z5, tool0;
	MoveL Offs(p0,54.0,29.0, 0), v10, z5, tool0;
	MoveL Offs(p0,54.0,28.0, 0), v10, z5, tool0;
	MoveL Offs(p0,53.0,28.0, 0), v10, z5, tool0;
	MoveL Offs(p0,51.0,25.0, 0), v10, z5, tool0;
	MoveL Offs(p0,51.0,25.0, 0), v10, z5, tool0;
	MoveL Offs(p0,51.0,24.0, 0), v10, z5, tool0;
	MoveL Offs(p0,51.0,23.0, 0), v10, z5, tool0;
	MoveL Offs(p0,52.0,23.0, 0), v10, z5, tool0;
	MoveL Offs(p0,52.0,23.0, 0), v10, z5, tool0;
	MoveL Offs(p0,53.0,22.0, 0), v10, z5, tool0;
	MoveL Offs(p0,54.0,22.0, 0), v10, z5, tool0;
	MoveL Offs(p0,57.0,22.0, 0), v10, z5, tool0;
	MoveL Offs(p0,58.0,22.0, 0), v10, z5, tool0;
	MoveL Offs(p0,59.0,22.0, 0), v10, z5, tool0;
	MoveL Offs(p0,59.0,22.0, 0), v10, z5, tool0;
	MoveL Offs(p0,60.0,22.0, 0), v10, z5, tool0;
	MoveL Offs(p0,62.0,22.0, 0), v10, z5, tool0;
	MoveL Offs(p0,63.0,23.0, 0), v10, z5, tool0;
	MoveL Offs(p0,65.0,22.0, 0), v10, z5, tool0;
	MoveL Offs(p0,66.0,22.0, 0), v10, z5, tool0;
	MoveL Offs(p0,66.0,21.0, 0), v10, z5, tool0;
	MoveL Offs(p0,67.0,20.0, 0), v10, z5, tool0;
	MoveL Offs(p0,69.0,18.0, 0), v10, z5, tool0;
	MoveL Offs(p0,67.0,18.0, 0), v10, z5, tool0;
	MoveL Offs(p0,64.0,18.0, 0), v10, z5, tool0;
	MoveL Offs(p0,63.0,18.0, 0), v10, z5, tool0;
	MoveL Offs(p0,62.0,17.0, 0), v10, z5, tool0;
	MoveL Offs(p0,61.0,17.0, 0), v10, z5, tool0;
	MoveL Offs(p0,60.0,17.0, 0), v10, z5, tool0;
	MoveL Offs(p0,59.0,16.0, 0), v10, z5, tool0;
	MoveL Offs(p0,58.0,16.0, 0), v10, z5, tool0;
	MoveL Offs(p0,57.0,16.0, 0), v10, z5, tool0;
	MoveL Offs(p0,55.0,14.0, 0), v10, z5, tool0;
	MoveL Offs(p0,54.0,14.0, 0), v10, z5, tool0;
	MoveL Offs(p0,54.0,13.0, 0), v10, z5, tool0;
	MoveL Offs(p0,53.0,13.0, 0), v10, z5, tool0;
	MoveL Offs(p0,53.0,13.0, 0), v10, z5, tool0;
	MoveL Offs(p0,51.0,11.0, 0), v10, z5, tool0;
	MoveL Offs(p0,50.0,12.0, 0), v10, z5, tool0;
	MoveL Offs(p0,49.0,15.0, 0), v10, z5, tool0;
	MoveL Offs(p0,49.0,17.0, 0), v10, z5, tool0;
	MoveL Offs(p0,49.0,18.0, 0), v10, z5, tool0;
	MoveL Offs(p0,48.0,20.0, 0), v10, z5, tool0;
	MoveL Offs(p0,48.0,21.0, 0), v10, z5, tool0;
	MoveL Offs(p0,48.0,23.0, 0), v10, z5, tool0;
	MoveL Offs(p0,49.0,24.0, 0), v10, z5, tool0;
	MoveL Offs(p0,49.0,25.0, 0), v10, z5, tool0;
	MoveL Offs(p0,49.0,26.0, 0), v10, z5, tool0;
	MoveL Offs(p0,50.0,29.0, 0), v10, z5, tool0;
	MoveL Offs(p0,50.0,29.0, 0), v10, z5, tool0;
	MoveL Offs(p0,51.0,29.0, 0), v10, z5, tool0;
	MoveL Offs(p0,51.0,30.0, 0), v10, z5, tool0;
	MoveL Offs(p0,51.0,30.0, 0), v10, z5, tool0;
	MoveL Offs(p0,53.0,33.0, 0), v10, z5, tool0;
	MoveL Offs(p0,54.0,33.0, 0), v10, z5, tool0;
	MoveL Offs(p0,56.0,34.0, 0), v10, z5, tool0;
	MoveL Offs(p0,57.0,35.0, 0), v10, z5, tool0;
	MoveL Offs(p0,58.0,35.0, 0), v10, z5, tool0;
	MoveL Offs(p0,59.0,36.0, 0), v10, z5, tool0;
	MoveL Offs(p0,60.0,36.0, 0), v10, z5, tool0;
	MoveL Offs(p0,61.0,36.0, 0), v10, z5, tool0;
	MoveL Offs(p0,61.0,34.0, 0), v10, z5, tool0;
	MoveJ Offs(p0,61.0,34.0, 20), v10, z1, tool0;
	MoveJ Offs(p0,102.0,31.0, 20), v10, z1, tool0;
	MoveJ Offs(p0,102.0,31.0, 0), v10, z1, tool0;
	MoveL Offs(p0,102.0,29.0, 0), v10, z5, tool0;
	MoveL Offs(p0,101.0,27.0, 0), v10, z5, tool0;
	MoveL Offs(p0,100.0,25.0, 0), v10, z5, tool0;
	MoveL Offs(p0,99.0,24.0, 0), v10, z5, tool0;
	MoveL Offs(p0,98.0,22.0, 0), v10, z5, tool0;
	MoveL Offs(p0,97.0,21.0, 0), v10, z5, tool0;
	MoveL Offs(p0,95.0,20.0, 0), v10, z5, tool0;
	MoveL Offs(p0,93.0,19.0, 0), v10, z5, tool0;
	MoveL Offs(p0,92.0,18.0, 0), v10, z5, tool0;
	MoveL Offs(p0,90.0,17.0, 0), v10, z5, tool0;
	MoveL Offs(p0,88.0,16.0, 0), v10, z5, tool0;
	MoveL Offs(p0,87.0,16.0, 0), v10, z5, tool0;
	MoveL Offs(p0,86.0,16.0, 0), v10, z5, tool0;
	MoveL Offs(p0,86.0,16.0, 0), v10, z5, tool0;
	MoveL Offs(p0,85.0,16.0, 0), v10, z5, tool0;
	MoveL Offs(p0,84.0,16.0, 0), v10, z5, tool0;
	MoveL Offs(p0,83.0,16.0, 0), v10, z5, tool0;
	MoveL Offs(p0,82.0,16.0, 0), v10, z5, tool0;
	MoveL Offs(p0,78.0,16.0, 0), v10, z5, tool0;
	MoveL Offs(p0,77.0,16.0, 0), v10, z5, tool0;
	MoveL Offs(p0,76.0,16.0, 0), v10, z5, tool0;
	MoveL Offs(p0,75.0,17.0, 0), v10, z5, tool0;
	MoveL Offs(p0,74.0,17.0, 0), v10, z5, tool0;
	MoveL Offs(p0,73.0,17.0, 0), v10, z5, tool0;
	MoveL Offs(p0,73.0,18.0, 0), v10, z5, tool0;
	MoveL Offs(p0,72.0,18.0, 0), v10, z5, tool0;
	MoveL Offs(p0,72.0,19.0, 0), v10, z5, tool0;
	MoveL Offs(p0,72.0,21.0, 0), v10, z5, tool0;
	MoveL Offs(p0,72.0,22.0, 0), v10, z5, tool0;
	MoveL Offs(p0,72.0,23.0, 0), v10, z5, tool0;
	MoveL Offs(p0,72.0,25.0, 0), v10, z5, tool0;
	MoveL Offs(p0,73.0,26.0, 0), v10, z5, tool0;
	MoveL Offs(p0,74.0,27.0, 0), v10, z5, tool0;
	MoveL Offs(p0,74.0,28.0, 0), v10, z5, tool0;
	MoveL Offs(p0,75.0,29.0, 0), v10, z5, tool0;
	MoveL Offs(p0,76.0,30.0, 0), v10, z5, tool0;
	MoveL Offs(p0,78.0,32.0, 0), v10, z5, tool0;
	MoveL Offs(p0,79.0,32.0, 0), v10, z5, tool0;
	MoveL Offs(p0,80.0,32.0, 0), v10, z5, tool0;
	MoveL Offs(p0,80.0,32.0, 0), v10, z5, tool0;
	MoveL Offs(p0,81.0,33.0, 0), v10, z5, tool0;
	MoveL Offs(p0,82.0,33.0, 0), v10, z5, tool0;
	MoveL Offs(p0,83.0,32.0, 0), v10, z5, tool0;
	MoveL Offs(p0,84.0,32.0, 0), v10, z5, tool0;
	MoveL Offs(p0,87.0,32.0, 0), v10, z5, tool0;
	MoveL Offs(p0,89.0,32.0, 0), v10, z5, tool0;
	MoveL Offs(p0,91.0,32.0, 0), v10, z5, tool0;
	MoveL Offs(p0,93.0,32.0, 0), v10, z5, tool0;
	MoveL Offs(p0,95.0,32.0, 0), v10, z5, tool0;
	MoveL Offs(p0,97.0,32.0, 0), v10, z5, tool0;
	MoveL Offs(p0,98.0,33.0, 0), v10, z5, tool0;
	MoveL Offs(p0,100.0,33.0, 0), v10, z5, tool0;
	MoveL Offs(p0,101.0,34.0, 0), v10, z5, tool0;
	MoveL Offs(p0,102.0,32.0, 0), v10, z5, tool0;
	MoveL Offs(p0,102.0,32.0, 0), v10, z5, tool0;
	MoveL Offs(p0,102.0,31.0, 0), v10, z5, tool0;
	MoveL Offs(p0,102.0,31.0, 0), v10, z5, tool0;
	MoveJ Offs(p0,102.0,31.0, 20), v10, z1, tool0;
	MoveJ Offs(p0,36.0,34.0, 20), v10, z1, tool0;
	MoveJ Offs(p0,36.0,34.0, 0), v10, z1, tool0;
	MoveL Offs(p0,38.0,34.0, 0), v10, z5, tool0;
	MoveL Offs(p0,39.0,33.0, 0), v10, z5, tool0;
	MoveL Offs(p0,39.0,33.0, 0), v10, z5, tool0;
	MoveL Offs(p0,39.0,33.0, 0), v10, z5, tool0;
	MoveL Offs(p0,41.0,32.0, 0), v10, z5, tool0;
	MoveL Offs(p0,39.0,31.0, 0), v10, z5, tool0;
	MoveL Offs(p0,36.0,29.0, 0), v10, z5, tool0;
	MoveL Offs(p0,36.0,29.0, 0), v10, z5, tool0;
	MoveL Offs(p0,35.0,28.0, 0), v10, z5, tool0;
	MoveL Offs(p0,35.0,27.0, 0), v10, z5, tool0;
	MoveL Offs(p0,34.0,27.0, 0), v10, z5, tool0;
	MoveL Offs(p0,34.0,26.0, 0), v10, z5, tool0;
	MoveL Offs(p0,33.0,26.0, 0), v10, z5, tool0;
	MoveL Offs(p0,31.0,25.0, 0), v10, z5, tool0;
	MoveL Offs(p0,29.0,26.0, 0), v10, z5, tool0;
	MoveL Offs(p0,28.0,26.0, 0), v10, z5, tool0;
	MoveL Offs(p0,27.0,26.0, 0), v10, z5, tool0;
	MoveL Offs(p0,26.0,26.0, 0), v10, z5, tool0;
	MoveL Offs(p0,26.0,26.0, 0), v10, z5, tool0;
	MoveL Offs(p0,25.0,26.0, 0), v10, z5, tool0;
	MoveL Offs(p0,25.0,26.0, 0), v10, z5, tool0;
	MoveL Offs(p0,24.0,26.0, 0), v10, z5, tool0;
	MoveL Offs(p0,25.0,22.0, 0), v10, z5, tool0;
	MoveL Offs(p0,25.0,21.0, 0), v10, z5, tool0;
	MoveL Offs(p0,26.0,20.0, 0), v10, z5, tool0;
	MoveL Offs(p0,27.0,20.0, 0), v10, z5, tool0;
	MoveL Offs(p0,27.0,19.0, 0), v10, z5, tool0;
	MoveL Offs(p0,28.0,19.0, 0), v10, z5, tool0;
	MoveL Offs(p0,29.0,18.0, 0), v10, z5, tool0;
	MoveL Offs(p0,30.0,16.0, 0), v10, z5, tool0;
	MoveL Offs(p0,31.0,15.0, 0), v10, z5, tool0;
	MoveL Offs(p0,31.0,13.0, 0), v10, z5, tool0;
	MoveL Offs(p0,31.0,13.0, 0), v10, z5, tool0;
	MoveL Offs(p0,31.0,12.0, 0), v10, z5, tool0;
	MoveL Offs(p0,31.0,12.0, 0), v10, z5, tool0;
	MoveL Offs(p0,31.0,12.0, 0), v10, z5, tool0;
	MoveL Offs(p0,31.0,11.0, 0), v10, z5, tool0;
	MoveL Offs(p0,30.0,12.0, 0), v10, z5, tool0;
	MoveL Offs(p0,28.0,13.0, 0), v10, z5, tool0;
	MoveL Offs(p0,27.0,13.0, 0), v10, z5, tool0;
	MoveL Offs(p0,27.0,13.0, 0), v10, z5, tool0;
	MoveL Offs(p0,26.0,14.0, 0), v10, z5, tool0;
	MoveL Offs(p0,25.0,14.0, 0), v10, z5, tool0;
	MoveL Offs(p0,25.0,14.0, 0), v10, z5, tool0;
	MoveL Offs(p0,24.0,14.0, 0), v10, z5, tool0;
	MoveL Offs(p0,23.0,14.0, 0), v10, z5, tool0;
	MoveL Offs(p0,21.0,14.0, 0), v10, z5, tool0;
	MoveL Offs(p0,20.0,16.0, 0), v10, z5, tool0;
	MoveL Offs(p0,20.0,20.0, 0), v10, z5, tool0;
	MoveL Offs(p0,20.0,22.0, 0), v10, z5, tool0;
	MoveL Offs(p0,20.0,24.0, 0), v10, z5, tool0;
	MoveL Offs(p0,21.0,26.0, 0), v10, z5, tool0;
	MoveL Offs(p0,21.0,28.0, 0), v10, z5, tool0;
	MoveL Offs(p0,22.0,29.0, 0), v10, z5, tool0;
	MoveL Offs(p0,24.0,31.0, 0), v10, z5, tool0;
	MoveL Offs(p0,25.0,32.0, 0), v10, z5, tool0;
	MoveL Offs(p0,27.0,33.0, 0), v10, z5, tool0;
	MoveL Offs(p0,30.0,34.0, 0), v10, z5, tool0;
	MoveL Offs(p0,30.0,34.0, 0), v10, z5, tool0;
	MoveL Offs(p0,31.0,34.0, 0), v10, z5, tool0;
	MoveL Offs(p0,32.0,35.0, 0), v10, z5, tool0;
	MoveL Offs(p0,33.0,35.0, 0), v10, z5, tool0;
	MoveL Offs(p0,34.0,35.0, 0), v10, z5, tool0;
	MoveL Offs(p0,35.0,34.0, 0), v10, z5, tool0;
	MoveL Offs(p0,36.0,34.0, 0), v10, z5, tool0;
	MoveL Offs(p0,36.0,34.0, 0), v10, z5, tool0;
	MoveJ Offs(p0,36.0,34.0, 20), v10, z1, tool0;
	MoveJ Offs(p0,15.0,33.0, 20), v10, z1, tool0;
	MoveJ Offs(p0,15.0,33.0, 0), v10, z1, tool0;
	MoveL Offs(p0,17.0,32.0, 0), v10, z5, tool0;
	MoveL Offs(p0,18.0,32.0, 0), v10, z5, tool0;
	MoveL Offs(p0,18.0,31.0, 0), v10, z5, tool0;
	MoveL Offs(p0,18.0,31.0, 0), v10, z5, tool0;
	MoveL Offs(p0,20.0,29.0, 0), v10, z5, tool0;
	MoveL Offs(p0,20.0,27.0, 0), v10, z5, tool0;
	MoveL Offs(p0,19.0,25.0, 0), v10, z5, tool0;
	MoveL Offs(p0,19.0,25.0, 0), v10, z5, tool0;
	MoveL Offs(p0,19.0,25.0, 0), v10, z5, tool0;
	MoveL Offs(p0,19.0,24.0, 0), v10, z5, tool0;
	MoveL Offs(p0,16.0,25.0, 0), v10, z5, tool0;
	MoveL Offs(p0,15.0,26.0, 0), v10, z5, tool0;
	MoveL Offs(p0,15.0,27.0, 0), v10, z5, tool0;
	MoveL Offs(p0,14.0,28.0, 0), v10, z5, tool0;
	MoveL Offs(p0,13.0,29.0, 0), v10, z5, tool0;
	MoveL Offs(p0,12.0,31.0, 0), v10, z5, tool0;
	MoveL Offs(p0,12.0,32.0, 0), v10, z5, tool0;
	MoveL Offs(p0,12.0,32.0, 0), v10, z5, tool0;
	MoveL Offs(p0,12.0,32.0, 0), v10, z5, tool0;
	MoveL Offs(p0,12.0,33.0, 0), v10, z5, tool0;
	MoveL Offs(p0,12.0,33.0, 0), v10, z5, tool0;
	MoveL Offs(p0,12.0,33.0, 0), v10, z5, tool0;
	MoveL Offs(p0,14.0,34.0, 0), v10, z5, tool0;
	MoveL Offs(p0,15.0,33.0, 0), v10, z5, tool0;
	MoveL Offs(p0,15.0,33.0, 0), v10, z5, tool0;
	MoveJ Offs(p0,15.0,33.0, 20), v10, z1, tool0;
	MoveJ Offs(p0,50.0,32.0, 20), v10, z1, tool0;
	MoveJ Offs(p0,50.0,32.0, 0), v10, z1, tool0;
	MoveL Offs(p0,50.0,32.0, 0), v10, z5, tool0;
	MoveL Offs(p0,50.0,30.0, 0), v10, z5, tool0;
	MoveL Offs(p0,48.0,28.0, 0), v10, z5, tool0;
	MoveL Offs(p0,46.0,27.0, 0), v10, z5, tool0;
	MoveL Offs(p0,45.0,27.0, 0), v10, z5, tool0;
	MoveL Offs(p0,42.0,26.0, 0), v10, z5, tool0;
	MoveL Offs(p0,41.0,26.0, 0), v10, z5, tool0;
	MoveL Offs(p0,39.0,25.0, 0), v10, z5, tool0;
	MoveL Offs(p0,38.0,24.0, 0), v10, z5, tool0;
	MoveL Offs(p0,37.0,24.0, 0), v10, z5, tool0;
	MoveL Offs(p0,36.0,23.0, 0), v10, z5, tool0;
	MoveL Offs(p0,36.0,22.0, 0), v10, z5, tool0;
	MoveL Offs(p0,36.0,21.0, 0), v10, z5, tool0;
	MoveL Offs(p0,36.0,20.0, 0), v10, z5, tool0;
	MoveL Offs(p0,38.0,19.0, 0), v10, z5, tool0;
	MoveL Offs(p0,39.0,18.0, 0), v10, z5, tool0;
	MoveL Offs(p0,40.0,18.0, 0), v10, z5, tool0;
	MoveL Offs(p0,41.0,18.0, 0), v10, z5, tool0;
	MoveL Offs(p0,42.0,18.0, 0), v10, z5, tool0;
	MoveL Offs(p0,45.0,17.0, 0), v10, z5, tool0;
	MoveL Offs(p0,46.0,17.0, 0), v10, z5, tool0;
	MoveL Offs(p0,46.0,17.0, 0), v10, z5, tool0;
	MoveL Offs(p0,46.0,17.0, 0), v10, z5, tool0;
	MoveL Offs(p0,47.0,17.0, 0), v10, z5, tool0;
	MoveL Offs(p0,47.0,17.0, 0), v10, z5, tool0;
	MoveL Offs(p0,47.0,17.0, 0), v10, z5, tool0;
	MoveL Offs(p0,48.0,15.0, 0), v10, z5, tool0;
	MoveL Offs(p0,49.0,13.0, 0), v10, z5, tool0;
	MoveL Offs(p0,49.0,13.0, 0), v10, z5, tool0;
	MoveL Offs(p0,49.0,13.0, 0), v10, z5, tool0;
	MoveL Offs(p0,49.0,12.0, 0), v10, z5, tool0;
	MoveL Offs(p0,49.0,12.0, 0), v10, z5, tool0;
	MoveL Offs(p0,46.0,12.0, 0), v10, z5, tool0;
	MoveL Offs(p0,45.0,12.0, 0), v10, z5, tool0;
	MoveL Offs(p0,44.0,12.0, 0), v10, z5, tool0;
	MoveL Offs(p0,42.0,11.0, 0), v10, z5, tool0;
	MoveL Offs(p0,40.0,11.0, 0), v10, z5, tool0;
	MoveL Offs(p0,39.0,11.0, 0), v10, z5, tool0;
	MoveL Offs(p0,37.0,10.0, 0), v10, z5, tool0;
	MoveL Offs(p0,36.0,10.0, 0), v10, z5, tool0;
	MoveL Offs(p0,35.0,10.0, 0), v10, z5, tool0;
	MoveL Offs(p0,33.0,11.0, 0), v10, z5, tool0;
	MoveL Offs(p0,33.0,12.0, 0), v10, z5, tool0;
	MoveL Offs(p0,32.0,12.0, 0), v10, z5, tool0;
	MoveL Offs(p0,32.0,13.0, 0), v10, z5, tool0;
	MoveL Offs(p0,32.0,14.0, 0), v10, z5, tool0;
	MoveL Offs(p0,32.0,14.0, 0), v10, z5, tool0;
	MoveL Offs(p0,32.0,17.0, 0), v10, z5, tool0;
	MoveL Offs(p0,32.0,18.0, 0), v10, z5, tool0;
	MoveL Offs(p0,32.0,19.0, 0), v10, z5, tool0;
	MoveL Offs(p0,32.0,20.0, 0), v10, z5, tool0;
	MoveL Offs(p0,32.0,21.0, 0), v10, z5, tool0;
	MoveL Offs(p0,33.0,22.0, 0), v10, z5, tool0;
	MoveL Offs(p0,33.0,22.0, 0), v10, z5, tool0;
	MoveL Offs(p0,33.0,23.0, 0), v10, z5, tool0;
	MoveL Offs(p0,35.0,26.0, 0), v10, z5, tool0;
	MoveL Offs(p0,36.0,26.0, 0), v10, z5, tool0;
	MoveL Offs(p0,37.0,27.0, 0), v10, z5, tool0;
	MoveL Offs(p0,37.0,28.0, 0), v10, z5, tool0;
	MoveL Offs(p0,38.0,29.0, 0), v10, z5, tool0;
	MoveL Offs(p0,39.0,29.0, 0), v10, z5, tool0;
	MoveL Offs(p0,40.0,30.0, 0), v10, z5, tool0;
	MoveL Offs(p0,41.0,30.0, 0), v10, z5, tool0;
	MoveL Offs(p0,43.0,31.0, 0), v10, z5, tool0;
	MoveL Offs(p0,43.0,31.0, 0), v10, z5, tool0;
	MoveL Offs(p0,44.0,31.0, 0), v10, z5, tool0;
	MoveL Offs(p0,45.0,32.0, 0), v10, z5, tool0;
	MoveL Offs(p0,46.0,32.0, 0), v10, z5, tool0;
	MoveL Offs(p0,46.0,32.0, 0), v10, z5, tool0;
	MoveL Offs(p0,47.0,32.0, 0), v10, z5, tool0;
	MoveL Offs(p0,48.0,32.0, 0), v10, z5, tool0;
	MoveL Offs(p0,50.0,32.0, 0), v10, z5, tool0;
	MoveJ Offs(p0,50.0,32.0, 20), v10, z1, tool0;
	MoveJ Offs(p0,63.0,25.0, 20), v10, z1, tool0;
	MoveJ Offs(p0,63.0,25.0, 0), v10, z1, tool0;
	MoveL Offs(p0,61.0,23.0, 0), v10, z5, tool0;
	MoveL Offs(p0,60.0,23.0, 0), v10, z5, tool0;
	MoveL Offs(p0,59.0,23.0, 0), v10, z5, tool0;
	MoveL Offs(p0,58.0,23.0, 0), v10, z5, tool0;
	MoveL Offs(p0,57.0,23.0, 0), v10, z5, tool0;
	MoveL Offs(p0,56.0,22.0, 0), v10, z5, tool0;
	MoveL Offs(p0,56.0,22.0, 0), v10, z5, tool0;
	MoveL Offs(p0,54.0,23.0, 0), v10, z5, tool0;
	MoveL Offs(p0,53.0,23.0, 0), v10, z5, tool0;
	MoveL Offs(p0,53.0,23.0, 0), v10, z5, tool0;
	MoveL Offs(p0,53.0,23.0, 0), v10, z5, tool0;
	MoveL Offs(p0,52.0,23.0, 0), v10, z5, tool0;
	MoveL Offs(p0,52.0,24.0, 0), v10, z5, tool0;
	MoveL Offs(p0,52.0,24.0, 0), v10, z5, tool0;
	MoveL Offs(p0,53.0,26.0, 0), v10, z5, tool0;
	MoveL Offs(p0,53.0,27.0, 0), v10, z5, tool0;
	MoveL Offs(p0,54.0,28.0, 0), v10, z5, tool0;
	MoveL Offs(p0,55.0,29.0, 0), v10, z5, tool0;
	MoveL Offs(p0,57.0,30.0, 0), v10, z5, tool0;
	MoveL Offs(p0,58.0,30.0, 0), v10, z5, tool0;
	MoveL Offs(p0,59.0,31.0, 0), v10, z5, tool0;
	MoveL Offs(p0,60.0,31.0, 0), v10, z5, tool0;
	MoveL Offs(p0,62.0,29.0, 0), v10, z5, tool0;
	MoveL Offs(p0,63.0,27.0, 0), v10, z5, tool0;
	MoveL Offs(p0,63.0,27.0, 0), v10, z5, tool0;
	MoveL Offs(p0,63.0,26.0, 0), v10, z5, tool0;
	MoveL Offs(p0,63.0,26.0, 0), v10, z5, tool0;
	MoveL Offs(p0,63.0,26.0, 0), v10, z5, tool0;
	MoveL Offs(p0,63.0,25.0, 0), v10, z5, tool0;
	MoveL Offs(p0,63.0,25.0, 0), v10, z5, tool0;
	MoveJ Offs(p0,63.0,25.0, 20), v10, z1, tool0;
	MoveJ Offs(p0,47.0,27.0, 20), v10, z1, tool0;
	MoveJ Offs(p0,47.0,27.0, 0), v10, z1, tool0;
	MoveL Offs(p0,47.0,23.0, 0), v10, z5, tool0;
	MoveL Offs(p0,47.0,23.0, 0), v10, z5, tool0;
	MoveL Offs(p0,47.0,22.0, 0), v10, z5, tool0;
	MoveL Offs(p0,47.0,22.0, 0), v10, z5, tool0;
